C01318=2036.464500,116.962000,-461.388800,-176.322032,-0.120321,-90.000210
C01319=2037.931200,116.962000,-461.158000,-176.322032,-0.120321,-90.000210
C01320=2041.746400,116.962000,-461.186100,-176.322032,-0.120321,-90.000210
C01321=2042.791200,116.962000,-462.109500,-176.322032,-0.120321,-90.000210
C01322=2046.669400,116.962000,-461.572000,-176.322032,-0.120321,-90.000210
C01323=2047.372600,116.962000,-461.209700,-176.322032,-0.120321,-90.000210
C01324=2051.683300,116.962000,-461.572800,-176.322032,-0.120321,-90.000210
C01325=2052.215000,116.962000,-461.119800,-176.322032,-0.120321,-90.000210
C01326=2053.341500,116.962000,-460.750600,-176.322032,-0.120321,-90.000210
C01327=2055.969200,116.962000,-461.503000,-176.322032,-0.120321,-90.000210
C01328=2057.527000,116.962000,-461.105400,-176.322032,-0.120321,-90.000210
C01329=2061.172200,116.962000,-461.573500,-176.322032,-0.120321,-90.000210
C01330=2062.439400,116.962000,-461.558500,-176.322032,-0.120321,-90.000210
C01331=2065.572800,116.962000,-461.680800,-176.322032,-0.120321,-90.000210
C01332=2067.063000,116.962000,-461.000200,-176.322032,-0.120321,-90.000210
C01333=2068.716200,116.962000,-461.083200,-176.322032,-0.120321,-90.000210
C01334=2071.053200,116.962000,-461.213900,-176.322032,-0.120321,-90.000210
C01335=2072.506400,116.962000,-461.300800,-176.322032,-0.120321,-90.000210
C01336=2074.891000,116.962000,-461.196800,-176.322032,-0.120321,-90.000210
C01337=2076.394800,116.962000,-460.759700,-176.322032,-0.120321,-90.000210
C01338=2078.471600,116.962000,-461.086200,-176.322032,-0.120321,-90.000210
C01339=2081.057100,116.962000,-461.349300,-176.322032,-0.120321,-90.000210
C01340=2082.319500,116.962000,-460.447100,-176.322032,-0.120321,-90.000210
C01341=2083.837500,116.962000,-461.092800,-176.322032,-0.120321,-90.000210
C01342=2086.755400,116.962000,-460.397000,-176.322032,-0.120321,-90.000210
C01343=2087.830400,116.962000,-460.548500,-176.322032,-0.120321,-90.000210
C01344=2091.095200,116.962000,-460.597700,-176.322032,-0.120321,-90.000210
C01345=2091.982300,116.962000,-460.859600,-176.322032,-0.120321,-90.000210
C01346=2095.305000,116.962000,-460.944600,-176.322032,-0.120321,-90.000210
C01347=2096.287900,116.962000,-460.453100,-176.322032,-0.120321,-90.000210
C01348=2100.115300,116.962000,-460.344000,-176.322032,-0.120321,-90.000210
C01349=2101.997500,116.962000,-459.946600,-176.322032,-0.120321,-90.000210
C01350=2105.324200,116.962000,-459.866500,-176.322032,-0.120321,-90.000210
C01351=2107.229200,116.962000,-459.869200,-176.322032,-0.120321,-90.000210
C01352=2110.594800,116.962000,-459.783900,-176.322032,-0.120321,-90.000210
C01353=2112.130300,116.962000,-459.809200,-176.322032,-0.120321,-90.000210
C01354=2116.276900,116.962000,-459.632100,-176.322032,-0.120321,-90.000210
C01355=2116.927300,116.962000,-459.418100,-176.322032,-0.120321,-90.000210
C01356=2120.552400,116.962000,-459.569000,-176.322032,-0.120321,-90.000210
C01357=2121.891800,116.962000,-459.359100,-176.322032,-0.120321,-90.000210
C01358=2125.448600,116.962000,-458.749300,-176.322032,-0.120321,-90.000210
C01359=2126.425900,116.962000,-458.730400,-176.322032,-0.120321,-90.000210
C01360=2130.843800,116.962000,-458.929300,-176.322032,-0.120321,-90.000210
C01361=2131.792200,116.962000,-458.786400,-176.322032,-0.120321,-90.000210
C01362=2136.497100,116.962000,-458.117400,-176.322032,-0.120321,-90.000210
C01363=2137.873200,116.962000,-458.357900,-176.322032,-0.120321,-90.000210
C01364=2141.381500,116.962000,-458.142600,-176.322032,-0.120321,-90.000210
C01365=2142.294300,116.962000,-457.951200,-176.322032,-0.120321,-90.000210
C01366=2144.907900,116.962000,-457.571500,-176.322032,-0.120321,-90.000210
C01367=2146.803600,116.962000,-457.969600,-176.322032,-0.120321,-90.000210
C01368=2150.305000,116.962000,-457.602500,-176.322032,-0.120321,-90.000210
C01369=2151.528700,116.962000,-457.480600,-176.322032,-0.120321,-90.000210
C01370=2155.429600,116.962000,-457.270200,-176.322032,-0.120321,-90.000210
C01371=2157.099200,116.962000,-457.023000,-176.322032,-0.120321,-90.000210
C01372=2160.581800,116.962000,-457.022500,-176.322032,-0.120321,-90.000210
C01373=2161.665200,116.962000,-457.050900,-176.322032,-0.120321,-90.000210
C01374=2166.487200,116.962000,-456.987300,-176.322032,-0.120321,-90.000210
C01375=2167.020300,116.962000,-456.749000,-176.322032,-0.120321,-90.000210
C01376=2171.823100,116.962000,-456.380100,-176.322032,-0.120321,-90.000210
C01377=2172.384000,116.962000,-456.372000,-176.322032,-0.120321,-90.000210
C01378=2176.071000,116.962000,-456.088800,-176.322032,-0.120321,-90.000210
C01379=2176.860800,116.962000,-456.069700,-176.322032,-0.120321,-90.000210
C01380=2178.404500,116.962000,-455.836200,-176.322032,-0.120321,-90.000210
C01381=2180.545900,116.962000,-456.078600,-176.322032,-0.120321,-90.000210
C01382=2181.385200,116.962000,-455.836400,-176.322032,-0.120321,-90.000210
C01383=2182.434900,116.962000,-455.383400,-176.322032,-0.120321,-90.000210
C01384=2183.123400,116.962000,-456.497400,-176.322032,-0.120321,-90.000210
C01385=2186.978500,116.962000,-454.141500,-176.322032,-0.120321,-90.000210
C01386=2187.489500,116.962000,-454.835800,-176.322032,-0.120321,-90.000210
C01387=2190.500600,116.962000,-454.234000,-176.322032,-0.120321,-90.000210
C01388=2187.460800,66.962000,-454.621100,-176.322032,-0.120321,-90.000210
C01389=2186.546200,66.962000,-454.703500,-176.322032,-0.120321,-90.000210
C01390=2183.293200,66.962000,-454.886900,-176.322032,-0.120321,-90.000210
C01391=2182.144700,66.962000,-455.103300,-176.322032,-0.120321,-90.000210
C01392=2179.703900,66.962000,-455.685400,-176.322032,-0.120321,-90.000210
C01393=2177.868100,66.962000,-455.661700,-176.322032,-0.120321,-90.000210
C01394=2176.413500,66.962000,-456.269000,-176.322032,-0.120321,-90.000210
C01395=2174.746100,66.962000,-455.981100,-176.322032,-0.120321,-90.000210
C01396=2172.146300,66.962000,-456.415800,-176.322032,-0.120321,-90.000210
C01397=2170.888100,66.962000,-456.236600,-176.322032,-0.120321,-90.000210
C01398=2167.524500,66.962000,-456.615100,-176.322032,-0.120321,-90.000210
C01399=2166.381300,66.962000,-456.924300,-176.322032,-0.120321,-90.000210
C01400=2162.140600,66.962000,-456.879000,-176.322032,-0.120321,-90.000210
C01401=2160.998700,66.962000,-457.154200,-176.322032,-0.120321,-90.000210
C01402=2157.715600,66.962000,-457.164000,-176.322032,-0.120321,-90.000210
C01403=2156.473800,66.962000,-457.185800,-176.322032,-0.120321,-90.000210
C01404=2152.943600,66.962000,-457.775400,-176.322032,-0.120321,-90.000210
C01405=2151.910000,66.962000,-457.828300,-176.322032,-0.120321,-90.000210
C01406=2147.641800,66.962000,-458.108900,-176.322032,-0.120321,-90.000210
C01407=2145.923200,66.962000,-458.251300,-176.322032,-0.120321,-90.000210
C01408=2142.640500,66.962000,-458.570300,-176.322032,-0.120321,-90.000210
C01409=2141.323600,66.962000,-458.433500,-176.322032,-0.120321,-90.000210
C01410=2137.209300,66.962000,-458.700300,-176.322032,-0.120321,-90.000210
C01411=2136.524600,66.962000,-458.900000,-176.322032,-0.120321,-90.000210
C01412=2132.513800,66.962000,-458.772000,-176.322032,-0.120321,-90.000210
C01413=2130.736700,66.962000,-459.053600,-176.322032,-0.120321,-90.000210
C01414=2126.998500,66.962000,-458.996300,-176.322032,-0.120321,-90.000210
C01415=2125.408700,66.962000,-459.180700,-176.322032,-0.120321,-90.000210
C01416=2122.103200,66.962000,-459.050100,-176.322032,-0.120321,-90.000210
C01417=2121.398500,66.962000,-459.543000,-176.322032,-0.120321,-90.000210
C01418=2117.274100,66.962000,-459.915900,-176.322032,-0.120321,-90.000210
C01419=2116.625200,66.962000,-459.803600,-176.322032,-0.120321,-90.000210
C01420=2112.741400,66.962000,-460.134900,-176.322032,-0.120321,-90.000210
C01421=2111.498800,66.962000,-459.901200,-176.322032,-0.120321,-90.000210
C01422=2107.364300,66.962000,-460.372100,-176.322032,-0.120321,-90.000210
C01423=2106.113400,66.962000,-460.172300,-176.322032,-0.120321,-90.000210
C01424=2102.272500,66.962000,-460.391900,-176.322032,-0.120321,-90.000210
C01425=2101.374900,66.962000,-460.360100,-176.322032,-0.120321,-90.000210
C01426=2097.664400,66.962000,-460.540100,-176.322032,-0.120321,-90.000210
C01427=2096.357700,66.962000,-460.242400,-176.322032,-0.120321,-90.000210
C01428=2092.441200,66.962000,-460.698100,-176.322032,-0.120321,-90.000210
C01429=2091.853500,66.962000,-460.725400,-176.322032,-0.120321,-90.000210
C01430=2090.580900,66.962000,-460.670300,-176.322032,-0.120321,-90.000210
C01431=2087.672500,66.962000,-460.988000,-176.322032,-0.120321,-90.000210
C01432=2086.891600,66.962000,-461.118100,-176.322032,-0.120321,-90.000210
C01433=2085.763200,66.962000,-461.022000,-176.322032,-0.120321,-90.000210
C01434=2082.853700,66.962000,-461.325900,-176.322032,-0.120321,-90.000210
C01435=2081.388800,66.962000,-461.142700,-176.322032,-0.120321,-90.000210
C01436=2078.659000,66.962000,-460.798200,-176.322032,-0.120321,-90.000210
C01437=2077.339900,66.962000,-460.592800,-176.322032,-0.120321,-90.000210
C01438=2076.693000,66.962000,-460.982800,-176.322032,-0.120321,-90.000210
C01439=2075.624700,66.962000,-460.685400,-176.322032,-0.120321,-90.000210
C01440=2072.957600,66.962000,-461.172700,-176.322032,-0.120321,-90.000210
C01441=2071.852900,66.962000,-461.354700,-176.322032,-0.120321,-90.000210
C01442=2068.101300,66.962000,-460.816200,-176.322032,-0.120321,-90.000210
C01443=2067.089500,66.962000,-461.221500,-176.322032,-0.120321,-90.000210
C01444=2066.067700,66.962000,-461.312200,-176.322032,-0.120321,-90.000210
C01445=2061.935200,66.962000,-461.790200,-176.322032,-0.120321,-90.000210
C01446=2061.303500,66.962000,-461.490200,-176.322032,-0.120321,-90.000210
C01447=2057.096300,66.962000,-461.766500,-176.322032,-0.120321,-90.000210
C01448=2056.220800,66.962000,-461.730600,-176.322032,-0.120321,-90.000210
C01449=2052.714800,66.962000,-461.821300,-176.322032,-0.120321,-90.000210
C01450=2051.615100,66.962000,-461.465000,-176.322032,-0.120321,-90.000210
C01451=2047.197100,66.962000,-462.015900,-176.322032,-0.120321,-90.000210
C01452=2046.669800,66.962000,-461.560700,-176.322032,-0.120321,-90.000210
C01453=2042.419200,66.962000,-461.438300,-176.322032,-0.120321,-90.000210
C01454=2041.321400,66.962000,-461.722900,-176.322032,-0.120321,-90.000210
C01455=2037.944000,66.962000,-461.891700,-176.322032,-0.120321,-90.000210
C01456=2036.779200,66.962000,-461.544600,-176.322032,-0.120321,-90.000210
C01457=2032.602700,66.962000,-461.671200,-176.322032,-0.120321,-90.000210
C01458=2032.128600,66.962000,-462.191800,-176.322032,-0.120321,-90.000210
C01459=2027.146500,66.962000,-461.876500,-176.322032,-0.120321,-90.000210
C01460=2026.533400,66.962000,-462.228000,-176.322032,-0.120321,-90.000210
C01461=2022.435100,66.962000,-462.037800,-176.322032,-0.120321,-90.000210
C01462=2021.425300,66.962000,-461.958100,-176.322032,-0.120321,-90.000210
C01463=2017.590500,66.962000,-461.902400,-176.322032,-0.120321,-90.000210
C01464=2017.006800,66.962000,-461.655800,-176.322032,-0.120321,-90.000210
C01465=2012.532100,66.962000,-462.194700,-176.322032,-0.120321,-90.000210
C01466=2012.154700,66.962000,-462.076800,-176.322032,-0.120321,-90.000210
C01467=2007.660100,66.962000,-462.120400,-176.322032,-0.120321,-90.000210
C01468=2006.639900,66.962000,-461.912600,-176.322032,-0.120321,-90.000210
C01469=2002.362600,66.962000,-462.269100,-176.322032,-0.120321,-90.000210
C01470=2001.731700,66.962000,-461.761800,-176.322032,-0.120321,-90.000210
C01471=1997.924200,66.962000,-462.524400,-176.322032,-0.120321,-90.000210
C01472=1996.573400,66.962000,-462.089000,-176.322032,-0.120321,-90.000210
C01473=1991.968800,66.962000,-462.726500,-176.322032,-0.120321,-90.000210
C01474=1991.298200,66.962000,-461.843300,-176.322032,-0.120321,-90.000210
C01475=1987.289200,66.962000,-461.999200,-176.322032,-0.120321,-90.000210
C01476=1986.814500,66.962000,-462.667300,-176.322032,-0.120321,-90.000210
C01477=1982.523900,66.962000,-462.299700,-176.322032,-0.120321,-90.000210
C01478=1981.365600,66.962000,-462.426300,-176.322032,-0.120321,-90.000210
C01479=1977.592200,66.962000,-462.407800,-176.322032,-0.120321,-90.000210
C01480=1976.591300,66.962000,-462.624200,-176.322032,-0.120321,-90.000210
C01481=1972.053400,66.962000,-462.402800,-176.322032,-0.120321,-90.000210
C01482=1971.187300,66.962000,-462.283800,-176.322032,-0.120321,-90.000210
C01483=1967.390600,66.962000,-462.352500,-176.322032,-0.120321,-90.000210
C01484=1966.281000,66.962000,-462.481700,-176.322032,-0.120321,-90.000210
C01485=1962.364900,66.962000,-462.681000,-176.322032,-0.120321,-90.000210
C01486=1961.526700,66.962000,-462.462900,-176.322032,-0.120321,-90.000210
C01487=1957.191000,66.962000,-462.718900,-176.322032,-0.120321,-90.000210
C01488=1956.508800,66.962000,-463.070800,-176.322032,-0.120321,-90.000210
C01489=1952.212400,66.962000,-462.659600,-176.322032,-0.120321,-90.000210
C01490=1951.195700,66.962000,-462.740300,-176.322032,-0.120321,-90.000210
C01491=1947.001000,66.962000,-462.695400,-176.322032,-0.120321,-90.000210
C01492=1946.188100,66.962000,-462.863100,-176.322032,-0.120321,-90.000210
C01493=1942.202500,66.962000,-462.673200,-176.322032,-0.120321,-90.000210
C01494=1941.556900,66.962000,-462.520400,-176.322032,-0.120321,-90.000210
C01495=1936.692100,66.962000,-462.898600,-176.322032,-0.120321,-90.000210
C01496=1936.108700,66.962000,-462.734800,-176.322032,-0.120321,-90.000210
C01497=1931.690400,66.962000,-462.982900,-176.322032,-0.120321,-90.000210
C01498=1930.845700,66.962000,-462.918100,-176.322032,-0.120321,-90.000210
C01499=1927.277900,66.962000,-463.021300,-176.322032,-0.120321,-90.000210
C01500=1926.380500,66.962000,-462.614200,-176.322032,-0.120321,-90.000210
C01501=1922.306400,66.962000,-462.887700,-176.322032,-0.120321,-90.000210
C01502=1920.906400,66.962000,-462.932600,-176.322032,-0.120321,-90.000210
C01503=1917.431300,66.962000,-462.524900,-176.322032,-0.120321,-90.000210
C01504=1916.235300,66.962000,-462.501100,-176.322032,-0.120321,-90.000210
C01505=1912.599900,66.962000,-462.603100,-176.322032,-0.120321,-90.000210
C01506=1910.569000,66.962000,-462.776000,-176.322032,-0.120321,-90.000210
C01507=1906.891700,66.962000,-462.472500,-176.322032,-0.120321,-90.000210
C01508=1905.947500,66.962000,-462.866000,-176.322032,-0.120321,-90.000210
C01509=1901.562100,66.962000,-462.900500,-176.322032,-0.120321,-90.000210
C01510=1901.024600,66.962000,-462.765600,-176.322032,-0.120321,-90.000210
C01511=1896.366700,66.962000,-462.571200,-176.322032,-0.120321,-90.000210
C01512=1895.945300,66.962000,-462.685500,-176.322032,-0.120321,-90.000210
C01513=1892.072500,66.962000,-462.600000,-176.322032,-0.120321,-90.000210
C01514=1887.540100,66.962000,-462.340500,-176.322032,-0.120321,-90.000210
C01515=1887.060500,66.962000,-462.329200,-176.322032,-0.120321,-90.000210
C01516=1883.578900,66.962000,-461.818100,-176.322032,-0.120321,-90.000210
C01517=1881.534600,66.962000,-462.313800,-176.322032,-0.120321,-90.000210
C01518=1877.920400,66.962000,-462.348400,-176.322032,-0.120321,-90.000210
C01519=1877.012100,66.962000,-462.257500,-176.322032,-0.120321,-90.000210
C01520=1873.176100,66.962000,-462.090200,-176.322032,-0.120321,-90.000210
C01521=1871.982100,66.962000,-461.820500,-176.322032,-0.120321,-90.000210
C01522=1867.738500,66.962000,-461.710300,-176.322032,-0.120321,-90.000210
C01523=1866.173600,66.962000,-461.878900,-176.322032,-0.120321,-90.000210
C01524=1862.125600,66.962000,-461.492800,-176.322032,-0.120321,-90.000210
C01525=1861.102200,66.962000,-461.128300,-176.322032,-0.120321,-90.000210
C01526=1858.018300,66.962000,-461.616900,-176.322032,-0.120321,-90.000210
C01527=1856.295800,66.962000,-460.869200,-176.322032,-0.120321,-90.000210
C01528=1854.579600,66.962000,-461.148100,-176.322032,-0.120321,-90.000210
C01529=1852.507200,66.962000,-461.287100,-176.322032,-0.120321,-90.000210
C01530=1851.208800,66.962000,-461.126800,-176.322032,-0.120321,-90.000210
C01531=1849.888800,66.962000,-460.848500,-176.322032,-0.120321,-90.000210
C01532=1847.630900,66.962000,-460.811400,-176.322032,-0.120321,-90.000210
C01533=1846.477100,66.962000,-460.758100,-176.322032,-0.120321,-90.000210
C01534=1844.129100,66.962000,-460.736500,-176.322032,-0.120321,-90.000210
C01535=1841.569400,66.962000,-460.494100,-176.322032,-0.120321,-90.000210
C01536=1837.832100,66.962000,-460.286000,-176.322032,-0.120321,-90.000210
C01537=1836.209500,66.962000,-460.222500,-176.322032,-0.120321,-90.000210
C01538=1832.383000,66.962000,-460.143800,-176.322032,-0.120321,-90.000210
C01539=1831.289100,66.962000,-459.907100,-176.322032,-0.120321,-90.000210
C01540=1827.422300,66.962000,-459.786000,-176.322032,-0.120321,-90.000210
C01541=1826.770000,66.962000,-459.789300,-176.322032,-0.120321,-90.000210
C01542=1822.655900,66.962000,-459.121000,-176.322032,-0.120321,-90.000210
C01543=1822.031800,66.962000,-459.340400,-176.322032,-0.120321,-90.000210
C01544=1817.166700,66.962000,-458.933700,-176.322032,-0.120321,-90.000210
C01545=1815.927200,66.962000,-458.829300,-176.322032,-0.120321,-90.000210
C01546=1812.134000,66.962000,-458.724000,-176.322032,-0.120321,-90.000210
C01547=1811.547400,66.962000,-458.669000,-176.322032,-0.120321,-90.000210
C01548=1807.539800,66.962000,-458.085800,-176.322032,-0.120321,-90.000210
C01549=1806.155800,66.962000,-458.104200,-176.322032,-0.120321,-90.000210
C01550=1802.582800,66.962000,-457.791500,-176.322032,-0.120321,-90.000210
C01551=1802.038800,66.962000,-457.763400,-176.322032,-0.120321,-90.000210
C01552=1797.104900,66.962000,-456.696100,-176.322032,-0.120321,-90.000210
C01553=1800.853000,16.962000,-457.600400,-176.322032,-0.120321,-90.000210
C01554=1801.833400,16.962000,-457.702300,-176.322032,-0.120321,-90.000210
C01555=1805.690500,16.962000,-457.850100,-176.322032,-0.120321,-90.000210
C01556=1806.955100,16.962000,-458.128800,-176.322032,-0.120321,-90.000210
C01557=1810.171000,16.962000,-458.514800,-176.322032,-0.120321,-90.000210
C01558=1812.204800,16.962000,-458.248700,-176.322032,-0.120321,-90.000210
C01559=1815.347500,16.962000,-458.808000,-176.322032,-0.120321,-90.000210
C01560=1816.625200,16.962000,-458.841700,-176.322032,-0.120321,-90.000210
C01561=1819.689800,16.962000,-458.842800,-176.322032,-0.120321,-90.000210
C01562=1821.724100,16.962000,-459.142000,-176.322032,-0.120321,-90.000210
C01563=1825.694700,16.962000,-459.364300,-176.322032,-0.120321,-90.000210
C01564=1826.988700,16.962000,-459.139000,-176.322032,-0.120321,-90.000210
C01565=1830.989300,16.962000,-460.055400,-176.322032,-0.120321,-90.000210
C01566=1832.117900,16.962000,-459.845800,-176.322032,-0.120321,-90.000210
C01567=1835.624600,16.962000,-460.233700,-176.322032,-0.120321,-90.000210
C01568=1836.819800,16.962000,-460.243900,-176.322032,-0.120321,-90.000210
C01569=1840.600200,16.962000,-460.486000,-176.322032,-0.120321,-90.000210
C01570=1841.684100,16.962000,-460.100000,-176.322032,-0.120321,-90.000210
C01571=1842.855500,16.962000,-460.996600,-176.322032,-0.120321,-90.000210
C01572=1846.207800,16.962000,-460.276800,-176.322032,-0.120321,-90.000210
C01573=1847.787400,16.962000,-460.089300,-176.322032,-0.120321,-90.000210
C01574=1850.604200,16.962000,-460.507100,-176.322032,-0.120321,-90.000210
C01575=1851.898200,16.962000,-460.731700,-176.322032,-0.120321,-90.000210
C01576=1853.812100,16.962000,-460.957800,-176.322032,-0.120321,-90.000210
C01577=1856.051100,16.962000,-461.225800,-176.322032,-0.120321,-90.000210
C01578=1856.992500,16.962000,-460.979300,-176.322032,-0.120321,-90.000210
C01579=1860.909800,16.962000,-460.744600,-176.322032,-0.120321,-90.000210
C01580=1862.312000,16.962000,-461.462200,-176.322032,-0.120321,-90.000210
C01581=1863.680400,16.962000,-461.168200,-176.322032,-0.120321,-90.000210
C01582=1867.087300,16.962000,-461.817800,-176.322032,-0.120321,-90.000210
C01583=1868.078400,16.962000,-460.823400,-176.322032,-0.120321,-90.000210
C01584=1871.197200,16.962000,-462.036800,-176.322032,-0.120321,-90.000210
C01585=1871.740000,16.962000,-461.205200,-176.322032,-0.120321,-90.000210
C01586=1876.026500,16.962000,-461.728400,-176.322032,-0.120321,-90.000210
C01587=1876.941400,16.962000,-461.824400,-176.322032,-0.120321,-90.000210
C01588=1879.389400,16.962000,-461.693700,-176.322032,-0.120321,-90.000210
C01589=1882.239000,16.962000,-461.511900,-176.322032,-0.120321,-90.000210
C01590=1883.592600,16.962000,-461.739600,-176.322032,-0.120321,-90.000210
C01591=1886.781000,16.962000,-462.128300,-176.322032,-0.120321,-90.000210
C01592=1888.118700,16.962000,-461.470900,-176.322032,-0.120321,-90.000210
C01593=1892.080400,16.962000,-462.546100,-176.322032,-0.120321,-90.000210
C01594=1893.191100,16.962000,-462.370500,-176.322032,-0.120321,-90.000210
C01595=1897.094800,16.962000,-462.092100,-176.322032,-0.120321,-90.000210
C01596=1898.386500,16.962000,-462.636900,-176.322032,-0.120321,-90.000210
C01597=1901.138700,16.962000,-462.159200,-176.322032,-0.120321,-90.000210
C01598=1902.847400,16.962000,-461.680000,-176.322032,-0.120321,-90.000210
C01599=1906.862100,16.962000,-462.063600,-176.322032,-0.120321,-90.000210
C01600=1907.774900,16.962000,-461.771400,-176.322032,-0.120321,-90.000210
C01601=1911.590400,16.962000,-461.818300,-176.322032,-0.120321,-90.000210
C01602=1916.132700,16.962000,-461.555400,-176.322032,-0.120321,-90.000210
C01603=1917.627600,16.962000,-462.395700,-176.322032,-0.120321,-90.000210
C01604=1920.150200,16.962000,-461.852400,-176.322032,-0.120321,-90.000210
C01605=1922.503800,16.962000,-462.108200,-176.322032,-0.120321,-90.000210
C01606=1925.787300,16.962000,-462.559600,-176.322032,-0.120321,-90.000210
C01607=1927.580300,16.962000,-462.489900,-176.322032,-0.120321,-90.000210
C01608=1930.883000,16.962000,-462.130700,-176.322032,-0.120321,-90.000210
C01609=1932.180200,16.962000,-462.049300,-176.322032,-0.120321,-90.000210
C01610=1936.098200,16.962000,-461.733900,-176.322032,-0.120321,-90.000210
C01611=1937.465400,16.962000,-461.859600,-176.322032,-0.120321,-90.000210
C01612=1940.869700,16.962000,-461.667300,-176.322032,-0.120321,-90.000210
C01613=1941.947000,16.962000,-461.985100,-176.322032,-0.120321,-90.000210
C01614=1946.026000,16.962000,-461.537600,-176.322032,-0.120321,-90.000210
C01615=1947.031900,16.962000,-460.749300,-176.322032,-0.120321,-90.000210
C01616=1950.520700,16.962000,-462.488400,-176.322032,-0.120321,-90.000210
C01617=1951.508200,16.962000,-462.017400,-176.322032,-0.120321,-90.000210
C01618=1953.630300,16.962000,-460.907700,-176.322032,-0.120321,-90.000210
C01619=1956.666900,16.962000,-461.810100,-176.322032,-0.120321,-90.000210
C01620=1958.240000,16.962000,-461.138900,-176.322032,-0.120321,-90.000210
C01621=1961.763500,16.962000,-461.648500,-176.322032,-0.120321,-90.000210
C01622=1962.592900,16.962000,-461.669800,-176.322032,-0.120321,-90.000210
C01623=1966.715800,16.962000,-462.226500,-176.322032,-0.120321,-90.000210
C01624=1967.742300,16.962000,-461.460300,-176.322032,-0.120321,-90.000210
C01625=1971.291200,16.962000,-461.488500,-176.322032,-0.120321,-90.000210
C01626=1972.357700,16.962000,-461.185800,-176.322032,-0.120321,-90.000210
C01627=1976.644300,16.962000,-461.744300,-176.322032,-0.120321,-90.000210
C01628=1977.172500,16.962000,-461.461900,-176.322032,-0.120321,-90.000210
C01629=1981.055200,16.962000,-462.223500,-176.322032,-0.120321,-90.000210
C01630=1982.924200,16.962000,-461.277500,-176.322032,-0.120321,-90.000210
C01631=1985.903600,16.962000,-461.979500,-176.322032,-0.120321,-90.000210
C01632=1987.027800,16.962000,-462.156500,-176.322032,-0.120321,-90.000210
C01633=1990.724500,16.962000,-461.454900,-176.322032,-0.120321,-90.000210
C01634=1991.847500,16.962000,-461.089000,-176.322032,-0.120321,-90.000210
C01635=1992.300200,16.962000,-461.929400,-176.322032,-0.120321,-90.000210
C01636=1995.887600,16.962000,-461.863300,-176.322032,-0.120321,-90.000210
C01637=1997.305400,16.962000,-462.410800,-176.322032,-0.120321,-90.000210
C01638=2001.335200,16.962000,-461.762900,-176.322032,-0.120321,-90.000210
C01639=2001.915900,16.962000,-461.490300,-176.322032,-0.120321,-90.000210
C01640=2003.087800,16.962000,-460.638700,-176.322032,-0.120321,-90.000210
C01641=2005.703100,16.962000,-462.013900,-176.322032,-0.120321,-90.000210
C01642=2007.016400,16.962000,-461.067600,-176.322032,-0.120321,-90.000210
C01643=2010.670700,16.962000,-461.084200,-176.322032,-0.120321,-90.000210
C01644=2011.764900,16.962000,-461.877300,-176.322032,-0.120321,-90.000210
C01645=2014.884300,16.962000,-460.917300,-176.322032,-0.120321,-90.000210
C01646=2017.022900,16.962000,-461.622600,-176.322032,-0.120321,-90.000210
C01647=2018.108600,16.962000,-461.481100,-176.322032,-0.120321,-90.000210
C01648=2020.072500,16.962000,-461.472200,-176.322032,-0.120321,-90.000210
C01649=2021.496700,16.962000,-461.126300,-176.322032,-0.120321,-90.000210
C01650=2022.573700,16.962000,-461.597500,-176.322032,-0.120321,-90.000210
C01651=2025.356300,16.962000,-460.919900,-176.322032,-0.120321,-90.000210
C01652=2027.389200,16.962000,-460.852400,-176.322032,-0.120321,-90.000210
C01653=2028.101900,16.962000,-461.298000,-176.322032,-0.120321,-90.000210
C01654=2031.703300,16.962000,-460.626700,-176.322032,-0.120321,-90.000210
C01655=2032.902100,16.962000,-461.367200,-176.322032,-0.120321,-90.000210
C01656=2035.802300,16.962000,-460.830300,-176.322032,-0.120321,-90.000210
C01657=2037.079400,16.962000,-460.852900,-176.322032,-0.120321,-90.000210
C01658=2038.174900,16.962000,-460.664800,-176.322032,-0.120321,-90.000210
C01659=2041.615300,16.962000,-461.220900,-176.322032,-0.120321,-90.000210
C01660=2042.295400,16.962000,-461.025900,-176.322032,-0.120321,-90.000210
C01661=2046.640700,16.962000,-460.294900,-176.322032,-0.120321,-90.000210
C01662=2047.090900,16.962000,-461.310000,-176.322032,-0.120321,-90.000210
C01663=2048.126700,16.962000,-461.431700,-176.322032,-0.120321,-90.000210
C01664=2051.137100,16.962000,-461.425400,-176.322032,-0.120321,-90.000210
C01665=2052.144900,16.962000,-460.788200,-176.322032,-0.120321,-90.000210
C01666=2053.757600,16.962000,-460.715100,-176.322032,-0.120321,-90.000210
C01667=2055.647100,16.962000,-461.029500,-176.322032,-0.120321,-90.000210
C01668=2056.837400,16.962000,-460.592600,-176.322032,-0.120321,-90.000210
C01669=2058.334000,16.962000,-460.769100,-176.322032,-0.120321,-90.000210
C01670=2060.286200,16.962000,-460.650500,-176.322032,-0.120321,-90.000210
C01671=2061.744300,16.962000,-461.198600,-176.322032,-0.120321,-90.000210
C01672=2063.209100,16.962000,-460.755400,-176.322032,-0.120321,-90.000210
C01673=2065.833000,16.962000,-461.205700,-176.322032,-0.120321,-90.000210
C01674=2067.142800,16.962000,-461.197800,-176.322032,-0.120321,-90.000210
C01675=2068.505600,16.962000,-461.026200,-176.322032,-0.120321,-90.000210
C01676=2071.236500,16.962000,-460.349100,-176.322032,-0.120321,-90.000210
C01677=2072.661000,16.962000,-460.841900,-176.322032,-0.120321,-90.000210
C01678=2073.832100,16.962000,-460.585700,-176.322032,-0.120321,-90.000210
C01679=2076.319000,16.962000,-460.985400,-176.322032,-0.120321,-90.000210
C01680=2077.381000,16.962000,-460.675300,-176.322032,-0.120321,-90.000210
C01681=2080.891400,16.962000,-460.532900,-176.322032,-0.120321,-90.000210
C01682=2081.908100,16.962000,-460.506000,-176.322032,-0.120321,-90.000210
C01683=2086.379400,16.962000,-460.673900,-176.322032,-0.120321,-90.000210
C01684=2087.105400,16.962000,-460.580200,-176.322032,-0.120321,-90.000210
C01685=2089.705100,16.962000,-460.365500,-176.322032,-0.120321,-90.000210
C01686=2091.207800,16.962000,-459.880700,-176.322032,-0.120321,-90.000210
C01687=2092.153100,16.962000,-461.155000,-176.322032,-0.120321,-90.000210
C01688=2096.423800,16.962000,-459.934900,-176.322032,-0.120321,-90.000210
C01689=2098.040400,16.962000,-460.150100,-176.322032,-0.120321,-90.000210
C01690=2101.854200,16.962000,-460.057700,-176.322032,-0.120321,-90.000210
C01691=2103.156700,16.962000,-459.863300,-176.322032,-0.120321,-90.000210
C01692=2107.026800,16.962000,-460.274800,-176.322032,-0.120321,-90.000210
C01693=2108.397300,16.962000,-459.836500,-176.322032,-0.120321,-90.000210
C01694=2111.487600,16.962000,-459.859600,-176.322032,-0.120321,-90.000210
C01695=2112.805300,16.962000,-459.587300,-176.322032,-0.120321,-90.000210
C01696=2116.598800,16.962000,-459.175700,-176.322032,-0.120321,-90.000210
C01697=2117.416700,16.962000,-459.383000,-176.322032,-0.120321,-90.000210
C01698=2121.547300,16.962000,-458.800000,-176.322032,-0.120321,-90.000210
C01699=2123.457300,16.962000,-458.872100,-176.322032,-0.120321,-90.000210
C01700=2126.573300,16.962000,-458.699900,-176.322032,-0.120321,-90.000210
C01701=2128.269900,16.962000,-458.632900,-176.322032,-0.120321,-90.000210
C01702=2132.065400,16.962000,-458.759400,-176.322032,-0.120321,-90.000210
C01703=2135.214800,16.962000,-458.605800,-176.322032,-0.120321,-90.000210
C01704=2137.412900,16.962000,-458.714700,-176.322032,-0.120321,-90.000210
C01705=2140.859300,16.962000,-458.398500,-176.322032,-0.120321,-90.000210
C01706=2142.455100,16.962000,-458.453300,-176.322032,-0.120321,-90.000210
C01707=2145.178200,16.962000,-458.252400,-176.322032,-0.120321,-90.000210
C01708=2146.847400,16.962000,-457.833500,-176.322032,-0.120321,-90.000210
C01709=2150.225600,16.962000,-458.008400,-176.322032,-0.120321,-90.000210
C01710=2151.796600,16.962000,-457.562300,-176.322032,-0.120321,-90.000210
C01711=2156.035700,16.962000,-457.211800,-176.322032,-0.120321,-90.000210
C01712=2157.040800,16.962000,-457.575900,-176.322032,-0.120321,-90.000210
C01713=2160.864800,16.962000,-456.858600,-176.322032,-0.120321,-90.000210
C01714=2162.183900,16.962000,-457.012700,-176.322032,-0.120321,-90.000210
C01715=2165.849300,16.962000,-456.622500,-176.322032,-0.120321,-90.000210
C01716=2166.839300,16.962000,-456.782400,-176.322032,-0.120321,-90.000210
C01717=2171.345200,16.962000,-456.357400,-176.322032,-0.120321,-90.000210
C01718=2172.133800,16.962000,-456.245200,-176.322032,-0.120321,-90.000210
C01719=2173.733600,16.962000,-455.771000,-176.322032,-0.120321,-90.000210
C01720=2176.308000,16.962000,-456.085000,-176.322032,-0.120321,-90.000210
C01721=2177.318900,16.962000,-456.012400,-176.322032,-0.120321,-90.000210
C01722=2178.967000,16.962000,-456.161600,-176.322032,-0.120321,-90.000210
C01723=2182.520600,16.962000,-455.315500,-176.322032,-0.120321,-90.000210
C01724=2183.036800,16.962000,-455.109100,-176.322032,-0.120321,-90.000210
C01725=2186.484700,16.962000,-454.724100,-176.322032,-0.120321,-90.000210
C01726=2187.838700,-33.038000,-454.194000,-176.322032,-0.120321,-90.000210
C01727=2186.454500,-33.038000,-454.700600,-176.322032,-0.120321,-90.000210
C01728=2183.213500,-33.038000,-455.001300,-176.322032,-0.120321,-90.000210
C01729=2181.860300,-33.038000,-455.251100,-176.322032,-0.120321,-90.000210
C01730=2179.250400,-33.038000,-455.735500,-176.322032,-0.120321,-90.000210
C01731=2176.946500,-33.038000,-456.101100,-176.322032,-0.120321,-90.000210
C01732=2175.426200,-33.038000,-456.242900,-176.322032,-0.120321,-90.000210
C01733=2172.831900,-33.038000,-455.920500,-176.322032,-0.120321,-90.000210
C01734=2171.322200,-33.038000,-456.459500,-176.322032,-0.120321,-90.000210
C01735=2168.024400,-33.038000,-456.212800,-176.322032,-0.120321,-90.000210
C01736=2167.233900,-33.038000,-456.321600,-176.322032,-0.120321,-90.000210
C01737=2165.443700,-33.038000,-456.078900,-176.322032,-0.120321,-90.000210
C01738=2162.061200,-33.038000,-456.737100,-176.322032,-0.120321,-90.000210
C01739=2160.812000,-33.038000,-456.592500,-176.322032,-0.120321,-90.000210
C01740=2157.031700,-33.038000,-457.063500,-176.322032,-0.120321,-90.000210
C01741=2155.682900,-33.038000,-456.848600,-176.322032,-0.120321,-90.000210
C01742=2152.307700,-33.038000,-457.399000,-176.322032,-0.120321,-90.000210
C01743=2151.095400,-33.038000,-456.909100,-176.322032,-0.120321,-90.000210
C01744=2147.119000,-33.038000,-457.698900,-176.322032,-0.120321,-90.000210
C01745=2146.285500,-33.038000,-457.464800,-176.322032,-0.120321,-90.000210
C01746=2142.094500,-33.038000,-457.317000,-176.322032,-0.120321,-90.000210
C01747=2140.940300,-33.038000,-458.102200,-176.322032,-0.120321,-90.000210
C01748=2137.249800,-33.038000,-457.849200,-176.322032,-0.120321,-90.000210
C01749=2135.800200,-33.038000,-458.404700,-176.322032,-0.120321,-90.000210
C01750=2132.447400,-33.038000,-457.888900,-176.322032,-0.120321,-90.000210
C01751=2130.881900,-33.038000,-458.017200,-176.322032,-0.120321,-90.000210
C01752=2127.696600,-33.038000,-458.392200,-176.322032,-0.120321,-90.000210
C01753=2125.934400,-33.038000,-457.589900,-176.322032,-0.120321,-90.000210
C01754=2122.034300,-33.038000,-458.169100,-176.322032,-0.120321,-90.000210
C01755=2120.860300,-33.038000,-458.711400,-176.322032,-0.120321,-90.000210
C01756=2116.693700,-33.038000,-459.001300,-176.322032,-0.120321,-90.000210
C01757=2115.536600,-33.038000,-458.957700,-176.322032,-0.120321,-90.000210
C01758=2112.057100,-33.038000,-458.432200,-176.322032,-0.120321,-90.000210
C01759=2111.520200,-33.038000,-458.485900,-176.322032,-0.120321,-90.000210
C01760=2107.335500,-33.038000,-459.507600,-176.322032,-0.120321,-90.000210
C01761=2106.856800,-33.038000,-458.373000,-176.322032,-0.120321,-90.000210
C01762=2102.696100,-33.038000,-458.762800,-176.322032,-0.120321,-90.000210
C01763=2101.749000,-33.038000,-459.833100,-176.322032,-0.120321,-90.000210
C01764=2097.182800,-33.038000,-459.129800,-176.322032,-0.120321,-90.000210
C01765=2095.888800,-33.038000,-459.330300,-176.322032,-0.120321,-90.000210
C01766=2091.851900,-33.038000,-459.415900,-176.322032,-0.120321,-90.000210
C01767=2091.217600,-33.038000,-459.772400,-176.322032,-0.120321,-90.000210
C01768=2087.288800,-33.038000,-459.756000,-176.322032,-0.120321,-90.000210
C01769=2085.837800,-33.038000,-458.509600,-176.322032,-0.120321,-90.000210
C01770=2081.795300,-33.038000,-459.414600,-176.322032,-0.120321,-90.000210
C01771=2080.997400,-33.038000,-459.367000,-176.322032,-0.120321,-90.000210
C01772=2076.630700,-33.038000,-458.860300,-176.322032,-0.120321,-90.000210
C01773=2076.051100,-33.038000,-459.656600,-176.322032,-0.120321,-90.000210
C01774=2072.015300,-33.038000,-458.713600,-176.322032,-0.120321,-90.000210
C01775=2071.035200,-33.038000,-459.399500,-176.322032,-0.120321,-90.000210
C01776=2067.236600,-33.038000,-459.249200,-176.322032,-0.120321,-90.000210
C01777=2065.839300,-33.038000,-458.730200,-176.322032,-0.120321,-90.000210
C01778=2062.160200,-33.038000,-458.971100,-176.322032,-0.120321,-90.000210
C01779=2061.058300,-33.038000,-459.739300,-176.322032,-0.120321,-90.000210
C01780=2057.081800,-33.038000,-459.848100,-176.322032,-0.120321,-90.000210
C01781=2055.954700,-33.038000,-459.049100,-176.322032,-0.120321,-90.000210
C01782=2051.778400,-33.038000,-459.442300,-176.322032,-0.120321,-90.000210
C01783=2051.093500,-33.038000,-460.698900,-176.322032,-0.120321,-90.000210
C01784=2047.182700,-33.038000,-460.243600,-176.322032,-0.120321,-90.000210
C01785=2046.729900,-33.038000,-459.904100,-176.322032,-0.120321,-90.000210
C01786=2042.216200,-33.038000,-460.457100,-176.322032,-0.120321,-90.000210
C01787=2041.294800,-33.038000,-458.744200,-176.322032,-0.120321,-90.000210
C01788=2037.518900,-33.038000,-459.148400,-176.322032,-0.120321,-90.000210
C01789=2035.474300,-33.038000,-460.335600,-176.322032,-0.120321,-90.000210
C01790=2031.929200,-33.038000,-460.110300,-176.322032,-0.120321,-90.000210
C01791=2029.976300,-33.038000,-459.700900,-176.322032,-0.120321,-90.000210
C01792=2027.239700,-33.038000,-459.399800,-176.322032,-0.120321,-90.000210
C01793=2025.810000,-33.038000,-459.211800,-176.322032,-0.120321,-90.000210
C01794=2021.686800,-33.038000,-459.299000,-176.322032,-0.120321,-90.000210
C01795=2021.017400,-33.038000,-460.534600,-176.322032,-0.120321,-90.000210
C01796=2016.905600,-33.038000,-459.977300,-176.322032,-0.120321,-90.000210
C01797=2012.348800,-33.038000,-459.566100,-176.322032,-0.120321,-90.000210
C01798=2011.690400,-33.038000,-460.454600,-176.322032,-0.120321,-90.000210
C01799=2008.176400,-33.038000,-460.018800,-176.322032,-0.120321,-90.000210
C01800=2006.344600,-33.038000,-459.093500,-176.322032,-0.120321,-90.000210
C01801=2003.207100,-33.038000,-460.862300,-176.322032,-0.120321,-90.000210
C01802=2002.338200,-33.038000,-459.942100,-176.322032,-0.120321,-90.000210
C01803=1999.720100,-33.038000,-461.131000,-176.322032,-0.120321,-90.000210
C01804=1997.072500,-33.038000,-460.970300,-176.322032,-0.120321,-90.000210
C01805=1996.611600,-33.038000,-458.972600,-176.322032,-0.120321,-90.000210
C01806=1991.746400,-33.038000,-460.075000,-176.322032,-0.120321,-90.000210
C01807=1990.974800,-33.038000,-458.928700,-176.322032,-0.120321,-90.000210
C01808=1988.250500,-33.038000,-460.146800,-176.322032,-0.120321,-90.000210
C01809=1986.586300,-33.038000,-459.666500,-176.322032,-0.120321,-90.000210
C01810=1982.669800,-33.038000,-460.393600,-176.322032,-0.120321,-90.000210
C01811=1982.006000,-33.038000,-460.568200,-176.322032,-0.120321,-90.000210
C01812=1978.599200,-33.038000,-461.372600,-176.322032,-0.120321,-90.000210
C01813=1977.058700,-33.038000,-459.119900,-176.322032,-0.120321,-90.000210
C01814=1975.657300,-33.038000,-460.292600,-176.322032,-0.120321,-90.000210
C01815=1971.969300,-33.038000,-459.202100,-176.322032,-0.120321,-90.000210
C01816=1970.572200,-33.038000,-461.094400,-176.322032,-0.120321,-90.000210
C01817=1967.981000,-33.038000,-460.591300,-176.322032,-0.120321,-90.000210
C01818=1966.614200,-33.038000,-459.028200,-176.322032,-0.120321,-90.000210
C01819=1962.506300,-33.038000,-459.253800,-176.322032,-0.120321,-90.000210
C01820=1961.381100,-33.038000,-459.030500,-176.322032,-0.120321,-90.000210
C01821=1959.432500,-33.038000,-461.204400,-176.322032,-0.120321,-90.000210
C01822=1957.002400,-33.038000,-460.734200,-176.322032,-0.120321,-90.000210
C01823=1956.020800,-33.038000,-460.682600,-176.322032,-0.120321,-90.000210
C01824=1952.100400,-33.038000,-459.585000,-176.322032,-0.120321,-90.000210
C01825=1951.434800,-33.038000,-460.976500,-176.322032,-0.120321,-90.000210
C01826=1947.466500,-33.038000,-460.666500,-176.322032,-0.120321,-90.000210
C01827=1946.943100,-33.038000,-460.699400,-176.322032,-0.120321,-90.000210
C01828=1945.653800,-33.038000,-461.235700,-176.322032,-0.120321,-90.000210
C01829=1943.038200,-33.038000,-460.079600,-176.322032,-0.120321,-90.000210
C01830=1941.410600,-33.038000,-459.356300,-176.322032,-0.120321,-90.000210
C01831=1937.364700,-33.038000,-460.486400,-176.322032,-0.120321,-90.000210
C01832=1936.135000,-33.038000,-459.630900,-176.322032,-0.120321,-90.000210
C01833=1932.447300,-33.038000,-460.184500,-176.322032,-0.120321,-90.000210
C01834=1931.839200,-33.038000,-460.658400,-176.322032,-0.120321,-90.000210
C01835=1928.033300,-33.038000,-459.392800,-176.322032,-0.120321,-90.000210
C01836=1926.449900,-33.038000,-459.869500,-176.322032,-0.120321,-90.000210
C01837=1922.847200,-33.038000,-459.598400,-176.322032,-0.120321,-90.000210
C01838=1922.331600,-33.038000,-460.286400,-176.322032,-0.120321,-90.000210
C01839=1921.130500,-33.038000,-461.293900,-176.322032,-0.120321,-90.000210
C01840=1917.493100,-33.038000,-460.855700,-176.322032,-0.120321,-90.000210
C01841=1916.540500,-33.038000,-460.962700,-176.322032,-0.120321,-90.000210
C01842=1912.790500,-33.038000,-461.250800,-176.322032,-0.120321,-90.000210
C01843=1911.355900,-33.038000,-460.108000,-176.322032,-0.120321,-90.000210
C01844=1907.391900,-33.038000,-460.981100,-176.322032,-0.120321,-90.000210
C01845=1906.312800,-33.038000,-459.849100,-176.322032,-0.120321,-90.000210
C01846=1903.183400,-33.038000,-459.145100,-176.322032,-0.120321,-90.000210
C01847=1902.901900,-33.038000,-461.310700,-176.322032,-0.120321,-90.000210
C01848=1900.636400,-33.038000,-460.740700,-176.322032,-0.120321,-90.000210
C01849=1897.837200,-33.038000,-460.909400,-176.322032,-0.120321,-90.000210
C01850=1897.597600,-33.038000,-459.241600,-176.322032,-0.120321,-90.000210
C01851=1894.765800,-33.038000,-461.260400,-176.322032,-0.120321,-90.000210
C01852=1892.524100,-33.038000,-459.593400,-176.322032,-0.120321,-90.000210
C01853=1891.819200,-33.038000,-460.231700,-176.322032,-0.120321,-90.000210
C01854=1887.245200,-33.038000,-461.384300,-176.322032,-0.120321,-90.000210
C01855=1886.571600,-33.038000,-459.789700,-176.322032,-0.120321,-90.000210
C01856=1884.738500,-33.038000,-461.008100,-176.322032,-0.120321,-90.000210
C01857=1882.108400,-33.038000,-460.748000,-176.322032,-0.120321,-90.000210
C01858=1880.397600,-33.038000,-459.760200,-176.322032,-0.120321,-90.000210
C01859=1876.965500,-33.038000,-461.214200,-176.322032,-0.120321,-90.000210
C01860=1876.113000,-33.038000,-460.611800,-176.322032,-0.120321,-90.000210
C01861=1872.874700,-33.038000,-460.371600,-176.322032,-0.120321,-90.000210
C01862=1871.807700,-33.038000,-460.314900,-176.322032,-0.120321,-90.000210
C01863=1868.205200,-33.038000,-461.054900,-176.322032,-0.120321,-90.000210
C01864=1866.817300,-33.038000,-458.988800,-176.322032,-0.120321,-90.000210
C01865=1866.123000,-33.038000,-460.006000,-176.322032,-0.120321,-90.000210
C01866=1861.764900,-33.038000,-459.510500,-176.322032,-0.120321,-90.000210
C01867=1861.028000,-33.038000,-460.387900,-176.322032,-0.120321,-90.000210
C01868=1856.776400,-33.038000,-458.848800,-176.322032,-0.120321,-90.000210
C01869=1855.827200,-33.038000,-460.033300,-176.322032,-0.120321,-90.000210
C01870=1851.961700,-33.038000,-459.904400,-176.322032,-0.120321,-90.000210
C01871=1850.635600,-33.038000,-459.546600,-176.322032,-0.120321,-90.000210
C01872=1846.693200,-33.038000,-459.808800,-176.322032,-0.120321,-90.000210
C01873=1846.101900,-33.038000,-459.693200,-176.322032,-0.120321,-90.000210
C01874=1842.005800,-33.038000,-458.706500,-176.322032,-0.120321,-90.000210
C01875=1840.272800,-33.038000,-458.341800,-176.322032,-0.120321,-90.000210
C01876=1836.351700,-33.038000,-458.618600,-176.322032,-0.120321,-90.000210
C01877=1835.877300,-33.038000,-459.666700,-176.322032,-0.120321,-90.000210
C01878=1831.732800,-33.038000,-458.830600,-176.322032,-0.120321,-90.000210
C01879=1827.627900,-33.038000,-458.623500,-176.322032,-0.120321,-90.000210
C01880=1827.146600,-33.038000,-458.251800,-176.322032,-0.120321,-90.000210
C01881=1822.666700,-33.038000,-457.936900,-176.322032,-0.120321,-90.000210
C01882=1821.003600,-33.038000,-458.961100,-176.322032,-0.120321,-90.000210
C01883=1817.553000,-33.038000,-458.342700,-176.322032,-0.120321,-90.000210
C01884=1816.574500,-33.038000,-457.949500,-176.322032,-0.120321,-90.000210
C01885=1812.646800,-33.038000,-458.310900,-176.322032,-0.120321,-90.000210
C01886=1811.813700,-33.038000,-458.144300,-176.322032,-0.120321,-90.000210
C01887=1807.630100,-33.038000,-457.924200,-176.322032,-0.120321,-90.000210
C01888=1806.662700,-33.038000,-457.994800,-176.322032,-0.120321,-90.000210
C01889=1802.325300,-33.038000,-457.304800,-176.322032,-0.120321,-90.000210
C01890=1801.377000,-33.038000,-457.525200,-176.322032,-0.120321,-90.000210
C01891=1797.263700,-83.038000,-456.540200,-176.322032,-0.120321,-90.000210
C01892=1801.377600,-83.038000,-456.423500,-176.322032,-0.120321,-90.000210
C01893=1802.039100,-83.038000,-456.528700,-176.322032,-0.120321,-90.000210
C01894=1806.137700,-83.038000,-456.420600,-176.322032,-0.120321,-90.000210
C01895=1807.517500,-83.038000,-457.040300,-176.322032,-0.120321,-90.000210
C01896=1811.510800,-83.038000,-457.342000,-176.322032,-0.120321,-90.000210
C01897=1812.761400,-83.038000,-456.921400,-176.322032,-0.120321,-90.000210
C01898=1816.633500,-83.038000,-456.944700,-176.322032,-0.120321,-90.000210
C01899=1818.180400,-83.038000,-456.446200,-176.322032,-0.120321,-90.000210
C01900=1821.418400,-83.038000,-457.315100,-176.322032,-0.120321,-90.000210
C01901=1822.147000,-83.038000,-457.631800,-176.322032,-0.120321,-90.000210
C01902=1825.940600,-83.038000,-457.200100,-176.322032,-0.120321,-90.000210
C01903=1827.184000,-83.038000,-456.413500,-176.322032,-0.120321,-90.000210
C01904=1831.431900,-83.038000,-456.952100,-176.322032,-0.120321,-90.000210
C01905=1832.943800,-83.038000,-457.695100,-176.322032,-0.120321,-90.000210
C01906=1836.336500,-83.038000,-456.649600,-176.322032,-0.120321,-90.000210
C01907=1837.917700,-83.038000,-456.259000,-176.322032,-0.120321,-90.000210
C01908=1841.653600,-83.038000,-456.294100,-176.322032,-0.120321,-90.000210
C01909=1842.500500,-83.038000,-457.453300,-176.322032,-0.120321,-90.000210
C01910=1846.655000,-83.038000,-456.158800,-176.322032,-0.120321,-90.000210
C01911=1847.914100,-83.038000,-456.971400,-176.322032,-0.120321,-90.000210
C01912=1850.886400,-83.038000,-457.947500,-176.322032,-0.120321,-90.000210
C01913=1851.924300,-83.038000,-456.455900,-176.322032,-0.120321,-90.000210
C01914=1853.746500,-83.038000,-455.909000,-176.322032,-0.120321,-90.000210
C01915=1856.801000,-83.038000,-456.540700,-176.322032,-0.120321,-90.000210
C01916=1857.226900,-83.038000,-457.572000,-176.322032,-0.120321,-90.000210
C01917=1861.661500,-83.038000,-457.096300,-176.322032,-0.120321,-90.000210
C01918=1862.298300,-83.038000,-456.125500,-176.322032,-0.120321,-90.000210
C01919=1866.796100,-83.038000,-456.521100,-176.322032,-0.120321,-90.000210
C01920=1868.461700,-83.038000,-457.691500,-176.322032,-0.120321,-90.000210
C01921=1871.614500,-83.038000,-458.087100,-176.322032,-0.120321,-90.000210
C01922=1872.861100,-83.038000,-457.346300,-176.322032,-0.120321,-90.000210
C01923=1876.567400,-83.038000,-457.369000,-176.322032,-0.120321,-90.000210
C01924=1877.660500,-83.038000,-456.269800,-176.322032,-0.120321,-90.000210
C01925=1881.048400,-83.038000,-455.876700,-176.322032,-0.120321,-90.000210
C01926=1882.363100,-83.038000,-456.205000,-176.322032,-0.120321,-90.000210
C01927=1885.185000,-83.038000,-458.324900,-176.322032,-0.120321,-90.000210
C01928=1886.931500,-83.038000,-457.616100,-176.322032,-0.120321,-90.000210
C01929=1891.295700,-83.038000,-456.342800,-176.322032,-0.120321,-90.000210
C01930=1892.497100,-83.038000,-456.878000,-176.322032,-0.120321,-90.000210
C01931=1895.995100,-83.038000,-455.878400,-176.322032,-0.120321,-90.000210
C01932=1897.742400,-83.038000,-457.729200,-176.322032,-0.120321,-90.000210
C01933=1901.249700,-83.038000,-458.023200,-176.322032,-0.120321,-90.000210
C01934=1902.218000,-83.038000,-457.070400,-176.322032,-0.120321,-90.000210
C01935=1904.345200,-83.038000,-456.433500,-176.322032,-0.120321,-90.000210
C01936=1906.979400,-83.038000,-457.295900,-176.322032,-0.120321,-90.000210
C01937=1909.333600,-83.038000,-458.869800,-176.322032,-0.120321,-90.000210
C01938=1911.531500,-83.038000,-456.868200,-176.322032,-0.120321,-90.000210
C01939=1912.668800,-83.038000,-456.031500,-176.322032,-0.120321,-90.000210
C01940=1916.918700,-83.038000,-458.426000,-176.322032,-0.120321,-90.000210
C01941=1917.701900,-83.038000,-457.524600,-176.322032,-0.120321,-90.000210
C01942=1922.078500,-83.038000,-458.064100,-176.322032,-0.120321,-90.000210
C01943=1922.918000,-83.038000,-457.294700,-176.322032,-0.120321,-90.000210
C01944=1926.700100,-83.038000,-459.205300,-176.322032,-0.120321,-90.000210
C01945=1927.250900,-83.038000,-457.182000,-176.322032,-0.120321,-90.000210
C01946=1931.982400,-83.038000,-456.069000,-176.322032,-0.120321,-90.000210
C01947=1932.147700,-83.038000,-457.389500,-176.322032,-0.120321,-90.000210
C01948=1936.037800,-83.038000,-455.685800,-176.322032,-0.120321,-90.000210
C01949=1937.405100,-83.038000,-458.998100,-176.322032,-0.120321,-90.000210
C01950=1940.796800,-83.038000,-456.815200,-176.322032,-0.120321,-90.000210
C01951=1942.395200,-83.038000,-457.390500,-176.322032,-0.120321,-90.000210
C01952=1944.845500,-83.038000,-458.958400,-176.322032,-0.120321,-90.000210
C01953=1946.875900,-83.038000,-456.942200,-176.322032,-0.120321,-90.000210
C01954=1950.220400,-83.038000,-456.395300,-176.322032,-0.120321,-90.000210
C01955=1951.914900,-83.038000,-457.328000,-176.322032,-0.120321,-90.000210
C01956=1955.423500,-83.038000,-456.371300,-176.322032,-0.120321,-90.000210
C01957=1956.995800,-83.038000,-458.267900,-176.322032,-0.120321,-90.000210
C01958=1959.602900,-83.038000,-456.606400,-176.322032,-0.120321,-90.000210
C01959=1961.519200,-83.038000,-458.740100,-176.322032,-0.120321,-90.000210
C01960=1965.354500,-83.038000,-457.213900,-176.322032,-0.120321,-90.000210
C01961=1966.905300,-83.038000,-455.640300,-176.322032,-0.120321,-90.000210
C01962=1971.058500,-83.038000,-457.727600,-176.322032,-0.120321,-90.000210
C01963=1972.264700,-83.038000,-456.054500,-176.322032,-0.120321,-90.000210
C01964=1974.115900,-83.038000,-455.778900,-176.322032,-0.120321,-90.000210
C01965=1976.905200,-83.038000,-457.645300,-176.322032,-0.120321,-90.000210
C01966=1977.676300,-83.038000,-458.975900,-176.322032,-0.120321,-90.000210
C01967=1981.825400,-83.038000,-457.787200,-176.322032,-0.120321,-90.000210
C01968=1983.003600,-83.038000,-456.479500,-176.322032,-0.120321,-90.000210
C01969=1986.886100,-83.038000,-458.067200,-176.322032,-0.120321,-90.000210
C01970=1989.294000,-83.038000,-455.376600,-176.322032,-0.120321,-90.000210
C01971=1992.332000,-83.038000,-457.244500,-176.322032,-0.120321,-90.000210
C01972=1994.263900,-83.038000,-458.489200,-176.322032,-0.120321,-90.000210
C01973=1996.329700,-83.038000,-458.739300,-176.322032,-0.120321,-90.000210
C01974=1997.462100,-83.038000,-458.441800,-176.322032,-0.120321,-90.000210
C01975=2001.519800,-83.038000,-456.471900,-176.322032,-0.120321,-90.000210
C01976=2002.039100,-83.038000,-458.226600,-176.322032,-0.120321,-90.000210
C01977=2006.365200,-83.038000,-457.899400,-176.322032,-0.120321,-90.000210
C01978=2007.611500,-83.038000,-456.940000,-176.322032,-0.120321,-90.000210
C01979=2011.393600,-83.038000,-457.792900,-176.322032,-0.120321,-90.000210
C01980=2012.219700,-83.038000,-456.288200,-176.322032,-0.120321,-90.000210
C01981=2015.812100,-83.038000,-458.440800,-176.322032,-0.120321,-90.000210
C01982=2017.030100,-83.038000,-456.217900,-176.322032,-0.120321,-90.000210
C01983=2021.279300,-83.038000,-458.175600,-176.322032,-0.120321,-90.000210
C01984=2022.237300,-83.038000,-456.596800,-176.322032,-0.120321,-90.000210
C01985=2026.020400,-83.038000,-457.311200,-176.322032,-0.120321,-90.000210
C01986=2026.631900,-83.038000,-456.498800,-176.322032,-0.120321,-90.000210
C01987=2030.724300,-83.038000,-456.286000,-176.322032,-0.120321,-90.000210
C01988=2031.361900,-83.038000,-458.301200,-176.322032,-0.120321,-90.000210
C01989=2035.954200,-83.038000,-458.269700,-176.322032,-0.120321,-90.000210
C01990=2037.154700,-83.038000,-456.120400,-176.322032,-0.120321,-90.000210
C01991=2038.215800,-83.038000,-455.719800,-176.322032,-0.120321,-90.000210
C01992=2042.068600,-83.038000,-457.753500,-176.322032,-0.120321,-90.000210
C01993=2043.184400,-83.038000,-456.910400,-176.322032,-0.120321,-90.000210
C01994=2046.139200,-83.038000,-458.371800,-176.322032,-0.120321,-90.000210
C01995=2046.949300,-83.038000,-456.269600,-176.322032,-0.120321,-90.000210
C01996=2051.275500,-83.038000,-458.065400,-176.322032,-0.120321,-90.000210
C01997=2052.389700,-83.038000,-458.406500,-176.322032,-0.120321,-90.000210
C01998=2056.771500,-83.038000,-457.622900,-176.322032,-0.120321,-90.000210
C01999=2057.436900,-83.038000,-456.230700,-176.322032,-0.120321,-90.000210
C02000=2061.046500,-83.038000,-458.471100,-176.322032,-0.120321,-90.000210
C02001=2062.307600,-83.038000,-458.250100,-176.322032,-0.120321,-90.000210
C02002=2066.484400,-83.038000,-456.692500,-176.322032,-0.120321,-90.000210
C02003=2067.746400,-83.038000,-456.025700,-176.322032,-0.120321,-90.000210
C02004=2069.633900,-83.038000,-456.869800,-176.322032,-0.120321,-90.000210
C02005=2071.554400,-83.038000,-455.892900,-176.322032,-0.120321,-90.000210
C02006=2072.633200,-83.038000,-457.582900,-176.322032,-0.120321,-90.000210
C02007=2076.333700,-83.038000,-457.344400,-176.322032,-0.120321,-90.000210
C02008=2077.954900,-83.038000,-457.572800,-176.322032,-0.120321,-90.000210
C02009=2081.587400,-83.038000,-458.305800,-176.322032,-0.120321,-90.000210
C02010=2082.795300,-83.038000,-457.300800,-176.322032,-0.120321,-90.000210
C02011=2086.722900,-83.038000,-457.167600,-176.322032,-0.120321,-90.000210
C02012=2088.396100,-83.038000,-455.635400,-176.322032,-0.120321,-90.000210
C02013=2091.369400,-83.038000,-457.029000,-176.322032,-0.120321,-90.000210
C02014=2092.142400,-83.038000,-456.409600,-176.322032,-0.120321,-90.000210
C02015=2096.407500,-83.038000,-457.112600,-176.322032,-0.120321,-90.000210
C02016=2098.017100,-83.038000,-456.330700,-176.322032,-0.120321,-90.000210
C02017=2101.502400,-83.038000,-456.888600,-176.322032,-0.120321,-90.000210
C02018=2102.273900,-83.038000,-457.221300,-176.322032,-0.120321,-90.000210
C02019=2106.143100,-83.038000,-455.631300,-176.322032,-0.120321,-90.000210
C02020=2106.749400,-83.038000,-456.158000,-176.322032,-0.120321,-90.000210
C02021=2109.791900,-83.038000,-455.916200,-176.322032,-0.120321,-90.000210
C02022=2112.245200,-83.038000,-457.240800,-176.322032,-0.120321,-90.000210
C02023=2113.650000,-83.038000,-456.224800,-176.322032,-0.120321,-90.000210
C02024=2116.592900,-83.038000,-457.485200,-176.322032,-0.120321,-90.000210
C02025=2118.171700,-83.038000,-457.734300,-176.322032,-0.120321,-90.000210
C02026=2121.489400,-83.038000,-455.713700,-176.322032,-0.120321,-90.000210
C02027=2123.002800,-83.038000,-456.620500,-176.322032,-0.120321,-90.000210
C02028=2126.272600,-83.038000,-456.458500,-176.322032,-0.120321,-90.000210
C02029=2127.021400,-83.038000,-456.241800,-176.322032,-0.120321,-90.000210
C02030=2130.380500,-83.038000,-455.975500,-176.322032,-0.120321,-90.000210
C02031=2131.517900,-83.038000,-456.490200,-176.322032,-0.120321,-90.000210
C02032=2133.000400,-83.038000,-457.288100,-176.322032,-0.120321,-90.000210
C02033=2136.544700,-83.038000,-456.314300,-176.322032,-0.120321,-90.000210
C02034=2137.561500,-83.038000,-456.582300,-176.322032,-0.120321,-90.000210
C02035=2140.485200,-83.038000,-456.953300,-176.322032,-0.120321,-90.000210
C02036=2142.027500,-83.038000,-455.560600,-176.322032,-0.120321,-90.000210
C02037=2143.171400,-83.038000,-455.414800,-176.322032,-0.120321,-90.000210
C02038=2146.645500,-83.038000,-455.859300,-176.322032,-0.120321,-90.000210
C02039=2147.458000,-83.038000,-455.621500,-176.322032,-0.120321,-90.000210
C02040=2151.204600,-83.038000,-456.511100,-176.322032,-0.120321,-90.000210
C02041=2152.489100,-83.038000,-455.289500,-176.322032,-0.120321,-90.000210
C02042=2156.219900,-83.038000,-454.624000,-176.322032,-0.120321,-90.000210
C02043=2157.348100,-83.038000,-456.405500,-176.322032,-0.120321,-90.000210
C02044=2160.882400,-83.038000,-455.794700,-176.322032,-0.120321,-90.000210
C02045=2161.954200,-83.038000,-456.106900,-176.322032,-0.120321,-90.000210
C02046=2164.616700,-83.038000,-456.092100,-176.322032,-0.120321,-90.000210
C02047=2167.074500,-83.038000,-455.772800,-176.322032,-0.120321,-90.000210
C02048=2168.424400,-83.038000,-455.258200,-176.322032,-0.120321,-90.000210
C02049=2171.813600,-83.038000,-455.571700,-176.322032,-0.120321,-90.000210
C02050=2173.005300,-83.038000,-455.054600,-176.322032,-0.120321,-90.000210
C02051=2176.119100,-83.038000,-455.289600,-176.322032,-0.120321,-90.000210
C02052=2177.224700,-83.038000,-454.727600,-176.322032,-0.120321,-90.000210
C02053=2181.520500,-83.038000,-454.439800,-176.322032,-0.120321,-90.000210
C02054=2182.514000,-83.038000,-455.350200,-176.322032,-0.120321,-90.000210
C02055=2185.997400,-83.038000,-454.048100,-176.322032,-0.120321,-90.000210
C02056=2187.456900,-83.038000,-453.822700,-176.322032,-0.120321,-90.000210
C02057=2187.373800,-133.038000,-453.058600,-176.322032,-0.120321,-90.000210
C02058=2186.173000,-133.038000,-452.904400,-176.322032,-0.120321,-90.000210
C02059=2181.970900,-133.038000,-453.572100,-176.322032,-0.120321,-90.000210
C02060=2181.086000,-133.038000,-452.259200,-176.322032,-0.120321,-90.000210
C02061=2177.642900,-133.038000,-452.841500,-176.322032,-0.120321,-90.000210
C02062=2176.178200,-133.038000,-454.289400,-176.322032,-0.120321,-90.000210
C02063=2172.448000,-133.038000,-453.722100,-176.322032,-0.120321,-90.000210
C02064=2171.093000,-133.038000,-454.267900,-176.322032,-0.120321,-90.000210
C02065=2167.273800,-133.038000,-452.746200,-176.322032,-0.120321,-90.000210
C02066=2166.588800,-133.038000,-454.231300,-176.322032,-0.120321,-90.000210
C02067=2162.219200,-133.038000,-453.252000,-176.322032,-0.120321,-90.000210
C02068=2161.345900,-133.038000,-454.239100,-176.322032,-0.120321,-90.000210
C02069=2157.321500,-133.038000,-453.888100,-176.322032,-0.120321,-90.000210
C02070=2156.881400,-133.038000,-454.395000,-176.322032,-0.120321,-90.000210
C02071=2152.391800,-133.038000,-453.025200,-176.322032,-0.120321,-90.000210
C02072=2151.094200,-133.038000,-453.392500,-176.322032,-0.120321,-90.000210
C02073=2147.436600,-133.038000,-454.712900,-176.322032,-0.120321,-90.000210
C02074=2146.105500,-133.038000,-452.489700,-176.322032,-0.120321,-90.000210
C02075=2142.728200,-133.038000,-453.775300,-176.322032,-0.120321,-90.000210
C02076=2141.248700,-133.038000,-452.540700,-176.322032,-0.120321,-90.000210
C02077=2137.222500,-133.038000,-454.428400,-176.322032,-0.120321,-90.000210
C02078=2135.926800,-133.038000,-452.055400,-176.322032,-0.120321,-90.000210
C02079=2132.036600,-133.038000,-454.675800,-176.322032,-0.120321,-90.000210
C02080=2131.072200,-133.038000,-452.371800,-176.322032,-0.120321,-90.000210
C02081=2127.231500,-133.038000,-454.577500,-176.322032,-0.120321,-90.000210
C02082=2126.719800,-133.038000,-455.046800,-176.322032,-0.120321,-90.000210
C02083=2122.286700,-133.038000,-454.057800,-176.322032,-0.120321,-90.000210
C02084=2120.565600,-133.038000,-454.499500,-176.322032,-0.120321,-90.000210
C02085=2117.277500,-133.038000,-451.748900,-176.322032,-0.120321,-90.000210
C02086=2115.704300,-133.038000,-454.725800,-176.322032,-0.120321,-90.000210
C02087=2112.314000,-133.038000,-455.309700,-176.322032,-0.120321,-90.000210
C02088=2111.374800,-133.038000,-454.773000,-176.322032,-0.120321,-90.000210
C02089=2106.960300,-133.038000,-454.636700,-176.322032,-0.120321,-90.000210
C02090=2106.224500,-133.038000,-451.947200,-176.322032,-0.120321,-90.000210
C02091=2102.475600,-133.038000,-454.889200,-176.322032,-0.120321,-90.000210
C02092=2101.684300,-133.038000,-454.016100,-176.322032,-0.120321,-90.000210
C02093=2097.394700,-133.038000,-453.504300,-176.322032,-0.120321,-90.000210
C02094=2096.126000,-133.038000,-453.711500,-176.322032,-0.120321,-90.000210
C02095=2092.164600,-133.038000,-454.984800,-176.322032,-0.120321,-90.000210
C02096=2091.068400,-133.038000,-453.204200,-176.322032,-0.120321,-90.000210
C02097=2087.539000,-133.038000,-454.995900,-176.322032,-0.120321,-90.000210
C02098=2086.319500,-133.038000,-453.344600,-176.322032,-0.120321,-90.000210
C02099=2082.211700,-133.038000,-452.721300,-176.322032,-0.120321,-90.000210
C02100=2081.793900,-133.038000,-455.285200,-176.322032,-0.120321,-90.000210
C02101=2076.871800,-133.038000,-455.786500,-176.322032,-0.120321,-90.000210
C02102=2075.480800,-133.038000,-454.697700,-176.322032,-0.120321,-90.000210
C02103=2071.132500,-133.038000,-452.233100,-176.322032,-0.120321,-90.000210
C02104=2068.360600,-133.038000,-453.353800,-176.322032,-0.120321,-90.000210
C02105=2066.886600,-133.038000,-454.523600,-176.322032,-0.120321,-90.000210
C02106=2063.419300,-133.038000,-454.885100,-176.322032,-0.120321,-90.000210
C02107=2061.568500,-133.038000,-455.500200,-176.322032,-0.120321,-90.000210
C02108=2057.624800,-133.038000,-455.500900,-176.322032,-0.120321,-90.000210
C02109=2057.004000,-133.038000,-454.887100,-176.322032,-0.120321,-90.000210
C02110=2053.191200,-133.038000,-453.109900,-176.322032,-0.120321,-90.000210
C02111=2051.756600,-133.038000,-455.206700,-176.322032,-0.120321,-90.000210
C02112=2048.678100,-133.038000,-455.166800,-176.322032,-0.120321,-90.000210
C02113=2047.198200,-133.038000,-451.334300,-176.322032,-0.120321,-90.000210
C02114=2043.365000,-133.038000,-453.901600,-176.322032,-0.120321,-90.000210
C02115=2041.721000,-133.038000,-453.658900,-176.322032,-0.120321,-90.000210
C02116=2037.967200,-133.038000,-452.938200,-176.322032,-0.120321,-90.000210
C02117=2036.885000,-133.038000,-452.406200,-176.322032,-0.120321,-90.000210
C02118=2032.344200,-133.038000,-453.994900,-176.322032,-0.120321,-90.000210
C02119=2031.784900,-133.038000,-453.270900,-176.322032,-0.120321,-90.000210
C02120=2028.013600,-133.038000,-454.885300,-176.322032,-0.120321,-90.000210
C02121=2026.752200,-133.038000,-451.706600,-176.322032,-0.120321,-90.000210
C02122=2022.750300,-133.038000,-452.672800,-176.322032,-0.120321,-90.000210
C02123=2021.130800,-133.038000,-454.197800,-176.322032,-0.120321,-90.000210
C02124=2018.221600,-133.038000,-456.075300,-176.322032,-0.120321,-90.000210
C02125=2016.328300,-133.038000,-454.195800,-176.322032,-0.120321,-90.000210
C02126=2012.311500,-133.038000,-453.970100,-176.322032,-0.120321,-90.000210
C02127=2011.246900,-133.038000,-455.091600,-176.322032,-0.120321,-90.000210
C02128=2007.556100,-133.038000,-454.730500,-176.322032,-0.120321,-90.000210
C02129=2006.472900,-133.038000,-455.380500,-176.322032,-0.120321,-90.000210
C02130=2001.970100,-133.038000,-452.315200,-176.322032,-0.120321,-90.000210
C02131=2000.601800,-133.038000,-455.368300,-176.322032,-0.120321,-90.000210
C02132=1997.453700,-133.038000,-454.754800,-176.322032,-0.120321,-90.000210
C02133=1996.489900,-133.038000,-453.154200,-176.322032,-0.120321,-90.000210
C02134=1992.029300,-133.038000,-454.096800,-176.322032,-0.120321,-90.000210
C02135=1991.548200,-133.038000,-453.439600,-176.322032,-0.120321,-90.000210
C02136=1986.869000,-133.038000,-453.776100,-176.322032,-0.120321,-90.000210
C02137=1985.820000,-133.038000,-453.951500,-176.322032,-0.120321,-90.000210
C02138=1982.350200,-133.038000,-453.250800,-176.322032,-0.120321,-90.000210
C02139=1981.268400,-133.038000,-454.339200,-176.322032,-0.120321,-90.000210
C02140=1977.068200,-133.038000,-455.258900,-176.322032,-0.120321,-90.000210
C02141=1976.165200,-133.038000,-454.760800,-176.322032,-0.120321,-90.000210
C02142=1972.187500,-133.038000,-453.934700,-176.322032,-0.120321,-90.000210
C02143=1971.166300,-133.038000,-454.891400,-176.322032,-0.120321,-90.000210
C02144=1967.473700,-133.038000,-454.101600,-176.322032,-0.120321,-90.000210
C02145=1966.060900,-133.038000,-455.392900,-176.322032,-0.120321,-90.000210
C02146=1961.675900,-133.038000,-454.814300,-176.322032,-0.120321,-90.000210
C02147=1961.012700,-133.038000,-452.894300,-176.322032,-0.120321,-90.000210
C02148=1956.743800,-133.038000,-453.982200,-176.322032,-0.120321,-90.000210
C02149=1956.343300,-133.038000,-454.968300,-176.322032,-0.120321,-90.000210
C02150=1952.013600,-133.038000,-454.486200,-176.322032,-0.120321,-90.000210
C02151=1951.398800,-133.038000,-454.244500,-176.322032,-0.120321,-90.000210
C02152=1947.484700,-133.038000,-455.723300,-176.322032,-0.120321,-90.000210
C02153=1946.181200,-133.038000,-453.128600,-176.322032,-0.120321,-90.000210
C02154=1942.188600,-133.038000,-455.373800,-176.322032,-0.120321,-90.000210
C02155=1941.485900,-133.038000,-456.084500,-176.322032,-0.120321,-90.000210
C02156=1937.171800,-133.038000,-452.942700,-176.322032,-0.120321,-90.000210
C02157=1936.777700,-133.038000,-454.336100,-176.322032,-0.120321,-90.000210
C02158=1932.595400,-133.038000,-454.888800,-176.322032,-0.120321,-90.000210
C02159=1931.693900,-133.038000,-455.408800,-176.322032,-0.120321,-90.000210
C02160=1927.858800,-133.038000,-454.821700,-176.322032,-0.120321,-90.000210
C02161=1926.659200,-133.038000,-452.831500,-176.322032,-0.120321,-90.000210
C02162=1922.429200,-133.038000,-455.521300,-176.322032,-0.120321,-90.000210
C02163=1921.791500,-133.038000,-455.397000,-176.322032,-0.120321,-90.000210
C02164=1918.851000,-133.038000,-454.800000,-176.322032,-0.120321,-90.000210
C02165=1917.010700,-133.038000,-452.245200,-176.322032,-0.120321,-90.000210
C02166=1914.019500,-133.038000,-455.955100,-176.322032,-0.120321,-90.000210
C02167=1912.257600,-133.038000,-454.967400,-176.322032,-0.120321,-90.000210
C02168=1910.541300,-133.038000,-455.157900,-176.322032,-0.120321,-90.000210
C02169=1907.346700,-133.038000,-452.907900,-176.322032,-0.120321,-90.000210
C02170=1905.944000,-133.038000,-455.678800,-176.322032,-0.120321,-90.000210
C02171=1902.008600,-133.038000,-455.767400,-176.322032,-0.120321,-90.000210
C02172=1901.152900,-133.038000,-455.565200,-176.322032,-0.120321,-90.000210
C02173=1897.458300,-133.038000,-453.701900,-176.322032,-0.120321,-90.000210
C02174=1896.226900,-133.038000,-455.974900,-176.322032,-0.120321,-90.000210
C02175=1892.459100,-133.038000,-454.184900,-176.322032,-0.120321,-90.000210
C02176=1891.454300,-133.038000,-455.045000,-176.322032,-0.120321,-90.000210
C02177=1887.301200,-133.038000,-455.639500,-176.322032,-0.120321,-90.000210
C02178=1887.094000,-133.038000,-454.789800,-176.322032,-0.120321,-90.000210
C02179=1881.707500,-133.038000,-454.831600,-176.322032,-0.120321,-90.000210
C02180=1880.935000,-133.038000,-454.177700,-176.322032,-0.120321,-90.000210
C02181=1877.465500,-133.038000,-455.617600,-176.322032,-0.120321,-90.000210
C02182=1876.452400,-133.038000,-453.948400,-176.322032,-0.120321,-90.000210
C02183=1872.152900,-133.038000,-453.644800,-176.322032,-0.120321,-90.000210
C02184=1871.251700,-133.038000,-454.462300,-176.322032,-0.120321,-90.000210
C02185=1867.034600,-133.038000,-455.314900,-176.322032,-0.120321,-90.000210
C02186=1866.363300,-133.038000,-454.623500,-176.322032,-0.120321,-90.000210
C02187=1861.762500,-133.038000,-454.870800,-176.322032,-0.120321,-90.000210
C02188=1860.357000,-133.038000,-454.604400,-176.322032,-0.120321,-90.000210
C02189=1856.822700,-133.038000,-454.995400,-176.322032,-0.120321,-90.000210
C02190=1855.793100,-133.038000,-453.836500,-176.322032,-0.120321,-90.000210
C02191=1852.369400,-133.038000,-454.282900,-176.322032,-0.120321,-90.000210
C02192=1851.706700,-133.038000,-454.546100,-176.322032,-0.120321,-90.000210
C02193=1847.013900,-133.038000,-454.673200,-176.322032,-0.120321,-90.000210
C02194=1846.392900,-133.038000,-456.104600,-176.322032,-0.120321,-90.000210
C02195=1842.853400,-133.038000,-454.701400,-176.322032,-0.120321,-90.000210
C02196=1841.764100,-133.038000,-455.566400,-176.322032,-0.120321,-90.000210
C02197=1837.893700,-133.038000,-456.110000,-176.322032,-0.120321,-90.000210
C02198=1836.646400,-133.038000,-454.832900,-176.322032,-0.120321,-90.000210
C02199=1834.854100,-133.038000,-455.757000,-176.322032,-0.120321,-90.000210
C02200=1831.290000,-133.038000,-454.943100,-176.322032,-0.120321,-90.000210
C02201=1827.575100,-133.038000,-455.770900,-176.322032,-0.120321,-90.000210
C02202=1826.678600,-133.038000,-455.706400,-176.322032,-0.120321,-90.000210
C02203=1825.333700,-133.038000,-455.274200,-176.322032,-0.120321,-90.000210
C02204=1822.107100,-133.038000,-455.697600,-176.322032,-0.120321,-90.000210
C02205=1821.345000,-133.038000,-456.237900,-176.322032,-0.120321,-90.000210
C02206=1819.592600,-133.038000,-456.016000,-176.322032,-0.120321,-90.000210
C02207=1817.152700,-133.038000,-456.207500,-176.322032,-0.120321,-90.000210
C02208=1815.752400,-133.038000,-456.162400,-176.322032,-0.120321,-90.000210
C02209=1812.473500,-133.038000,-455.878000,-176.322032,-0.120321,-90.000210
C02210=1811.262800,-133.038000,-455.512600,-176.322032,-0.120321,-90.000210
C02211=1807.875800,-133.038000,-456.284700,-176.322032,-0.120321,-90.000210
C02212=1807.109300,-133.038000,-456.069700,-176.322032,-0.120321,-90.000210
C02213=1805.572300,-133.038000,-455.935000,-176.322032,-0.120321,-90.000210
C02214=1802.605100,-133.038000,-455.813800,-176.322032,-0.120321,-90.000210
C02215=1801.855500,-133.038000,-456.078200,-176.322032,-0.120321,-90.000210
C02216=1800.000800,-133.038000,-456.024600,-176.322032,-0.120321,-90.000210
C02217=1796.212400,-133.038000,-456.323000,-176.322032,-0.120321,-90.000210
C02218=1811.635000,221.108300,-503.720300,90.647653,-0.183346,-0.000000
C02219=2127.176000,221.135000,-503.720300,90.647653,-0.183346,-0.000000
C02220=2158.549300,221.162700,-503.720300,90.647653,-0.183346,-0.000000
C02221=1815.760400,221.193100,-503.720300,90.647653,-0.183346,-0.000000
C02222=1821.263900,221.224800,-503.720300,90.647653,-0.183346,-0.000000
C02223=1812.312200,221.239900,-503.720300,90.647653,-0.183346,-0.000000
C02224=1809.093700,221.252000,-503.720300,90.647653,-0.183346,-0.000000
C02225=1831.237900,221.270100,-503.720300,90.647653,-0.183346,-0.000000
C02226=1825.910000,221.290400,-503.720300,90.647653,-0.183346,-0.000000
C02227=1834.967300,221.302200,-503.720300,90.647653,-0.183346,-0.000000
C02228=1839.702600,221.325900,-503.720300,90.647653,-0.183346,-0.000000
C02229=1835.410300,221.337300,-503.720300,90.647653,-0.183346,-0.000000
C02230=2118.838500,221.344100,-503.720300,90.647653,-0.183346,-0.000000
C02231=2151.568300,221.348800,-503.720300,90.647653,-0.183346,-0.000000
C02232=2174.762900,221.357600,-503.720300,90.647653,-0.183346,-0.000000
C02233=1808.009800,221.388700,-503.720300,90.647653,-0.183346,-0.000000
C02234=2144.201400,221.400900,-503.720300,90.647653,-0.183346,-0.000000
C02235=1798.112100,221.410000,-503.720300,90.647653,-0.183346,-0.000000
C02236=1837.822200,221.419800,-503.720300,90.647653,-0.183346,-0.000000
C02237=2112.433200,221.443100,-503.720300,90.647653,-0.183346,-0.000000
C02238=2136.213500,221.451500,-503.720300,90.647653,-0.183346,-0.000000
C02239=2089.573900,221.466700,-503.720300,90.647653,-0.183346,-0.000000
C02240=1866.266000,221.478900,-503.720300,90.647653,-0.183346,-0.000000
C02241=2119.282900,221.493800,-503.720300,90.647653,-0.183346,-0.000000
C02242=1857.771200,221.511800,-503.720300,90.647653,-0.183346,-0.000000
C02243=2166.291900,221.526500,-503.720300,90.647653,-0.183346,-0.000000
C02244=1850.974600,221.541100,-503.720300,90.647653,-0.183346,-0.000000
C02245=2143.673000,221.556300,-503.720300,90.647653,-0.183346,-0.000000
C02246=1828.630300,221.583500,-503.720300,90.647653,-0.183346,-0.000000
C02247=1860.958700,221.587300,-503.720300,90.647653,-0.183346,-0.000000
C02248=2184.435100,221.597500,-503.720300,90.647653,-0.183346,-0.000000
C02249=2090.804900,221.609300,-503.720300,90.647653,-0.183346,-0.000000
C02250=1817.450100,221.621800,-503.720300,90.647653,-0.183346,-0.000000
C02251=2128.070000,221.637700,-503.720300,90.647653,-0.183346,-0.000000
C02252=2189.176300,221.647500,-503.720300,90.647653,-0.183346,-0.000000
C02253=2117.034000,221.655300,-503.720300,90.647653,-0.183346,-0.000000
C02254=2108.809800,221.660300,-503.720300,90.647653,-0.183346,-0.000000
C02255=2089.962200,221.676200,-503.720300,90.647653,-0.183346,-0.000000
C02256=2113.622500,221.682600,-503.720300,90.647653,-0.183346,-0.000000
C02257=2125.630600,221.687300,-503.720300,90.647653,-0.183346,-0.000000
C02258=2088.737700,221.698800,-503.720300,90.647653,-0.183346,-0.000000
C02259=1865.593300,221.709000,-503.720300,90.647653,-0.183346,-0.000000
C02260=2127.249600,221.720500,-503.720300,90.647653,-0.183346,-0.000000
C02261=2081.446100,221.733300,-503.720300,90.647653,-0.183346,-0.000000
C02262=2078.914800,221.740800,-503.720300,90.647653,-0.183346,-0.000000
C02263=1876.021100,221.753900,-503.720300,90.647653,-0.183346,-0.000000
C02264=1875.515000,221.766700,-503.720300,90.647653,-0.183346,-0.000000
C02265=2183.148600,221.795100,-503.720300,90.647653,-0.183346,-0.000000
C02266=2072.022500,221.806300,-503.720300,90.647653,-0.183346,-0.000000
C02267=2079.695800,221.820800,-503.720300,90.647653,-0.183346,-0.000000
C02268=1887.088100,221.832300,-503.720300,90.647653,-0.183346,-0.000000
C02269=2188.540200,221.850500,-503.720300,90.647653,-0.183346,-0.000000
C02270=2075.988300,221.856300,-503.720300,90.647653,-0.183346,-0.000000
C02271=2063.126900,221.863400,-503.720300,90.647653,-0.183346,-0.000000
C02272=1880.005300,221.883000,-503.720300,90.647653,-0.183346,-0.000000
C02273=2072.176800,221.892200,-503.720300,90.647653,-0.183346,-0.000000
C02274=2142.155500,221.923200,-503.720300,90.647653,-0.183346,-0.000000
C02275=2163.272300,221.942100,-503.720300,90.647653,-0.183346,-0.000000
C02276=2043.282500,221.953200,-503.720300,90.647653,-0.183346,-0.000000
C02277=2143.086100,221.981600,-503.720300,90.647653,-0.183346,-0.000000
C02278=2151.779800,221.997200,-503.720300,90.647653,-0.183346,-0.000000
C02279=1889.947900,222.011300,-503.720300,90.647653,-0.183346,-0.000000
C02280=2187.503800,222.024700,-503.720300,90.647653,-0.183346,-0.000000
C02281=1997.220300,222.037400,-503.720300,90.647653,-0.183346,-0.000000
C02282=1908.585700,222.055600,-503.720300,90.647653,-0.183346,-0.000000
C02283=1902.103800,222.075200,-503.720300,90.647653,-0.183346,-0.000000
C02284=1894.253500,222.092100,-503.720300,90.647653,-0.183346,-0.000000
C02285=2087.902000,222.095600,-503.720300,90.647653,-0.183346,-0.000000
C02286=1918.899200,222.119100,-503.720300,90.647653,-0.183346,-0.000000
C02287=1997.786400,222.136500,-503.720300,90.647653,-0.183346,-0.000000
C02288=1996.583100,222.154600,-503.720300,90.647653,-0.183346,-0.000000
C02289=1985.344900,222.169500,-503.720300,90.647653,-0.183346,-0.000000
C02290=1910.038100,222.180600,-503.720300,90.647653,-0.183346,-0.000000
C02291=2048.549000,222.196100,-503.720300,90.647653,-0.183346,-0.000000
C02292=2035.591900,222.207300,-503.720300,90.647653,-0.183346,-0.000000
C02293=2032.094500,222.238400,-503.720300,90.647653,-0.183346,-0.000000
C02294=1901.470500,222.247800,-503.720300,90.647653,-0.183346,-0.000000
C02295=1911.640600,222.265500,-503.720300,90.647653,-0.183346,-0.000000
C02296=2025.335900,222.272500,-503.720300,90.647653,-0.183346,-0.000000
C02297=1897.938300,222.297800,-503.720300,90.647653,-0.183346,-0.000000
C02298=2028.686800,222.312700,-503.720300,90.647653,-0.183346,-0.000000
C02299=1901.595600,222.321100,-503.720300,90.647653,-0.183346,-0.000000
C02300=1927.085400,222.331600,-503.720300,90.647653,-0.183346,-0.000000
C02301=2002.627400,222.354900,-503.720300,90.647653,-0.183346,-0.000000
C02302=1981.632500,222.370800,-503.720300,90.647653,-0.183346,-0.000000
C02303=2008.400500,222.382000,-503.720300,90.647653,-0.183346,-0.000000
C02304=2016.963500,222.395500,-503.720300,90.647653,-0.183346,-0.000000
C02305=1927.753100,222.407300,-503.720300,90.647653,-0.183346,-0.000000
C02306=1936.624300,222.421800,-503.720300,90.647653,-0.183346,-0.000000
C02307=1941.897200,222.437700,-503.720300,90.647653,-0.183346,-0.000000
C02308=1915.919800,222.454300,-503.720300,90.647653,-0.183346,-0.000000
C02309=1941.539300,222.475200,-503.720300,90.647653,-0.183346,-0.000000
C02310=1969.735800,222.506600,-503.720300,90.647653,-0.183346,-0.000000
C02311=1958.400500,222.542400,-503.720300,90.647653,-0.183346,-0.000000
C02312=1952.915100,222.559000,-503.720300,90.647653,-0.183346,-0.000000
C02313=1927.316500,222.576200,-503.720300,90.647653,-0.183346,-0.000000
C02314=1935.896700,222.598500,-503.720300,90.647653,-0.183346,-0.000000
C02315=1927.083400,222.622300,-503.720300,90.647653,-0.183346,-0.000000
C02316=1971.501900,222.663700,-503.720300,90.647653,-0.183346,-0.000000
C02317=1985.419500,222.704600,-503.720300,90.647653,-0.183346,-0.000000
C02318=1933.249300,222.721700,-503.720300,90.647653,-0.183346,-0.000000
C02319=1983.244600,222.757300,-503.720300,90.647653,-0.183346,-0.000000
C02320=1966.958500,222.772500,-503.720300,90.647653,-0.183346,-0.000000
C02321=1971.033000,222.798900,-503.720300,90.647653,-0.183346,-0.000000
C02322=1977.908800,222.826200,-503.720300,90.647653,-0.183346,-0.000000
C02323=1956.249600,222.922500,-503.720300,90.647653,-0.183346,-0.000000
C02324=1963.733300,222.913400,-553.720300,90.647653,-0.183346,-0.000000
C02325=1956.256400,222.869900,-553.720300,90.647653,-0.183346,-0.000000
C02326=1948.604000,222.845500,-553.720300,90.647653,-0.183346,-0.000000
C02327=1964.013100,222.822500,-553.720300,90.647653,-0.183346,-0.000000
C02328=1979.543200,222.774200,-553.720300,90.647653,-0.183346,-0.000000
C02329=1979.134100,222.749900,-553.720300,90.647653,-0.183346,-0.000000
C02330=1991.483000,222.727900,-553.720300,90.647653,-0.183346,-0.000000
C02331=1961.051700,222.704900,-553.720300,90.647653,-0.183346,-0.000000
C02332=1983.390700,222.687000,-553.720300,90.647653,-0.183346,-0.000000
C02333=1962.251800,222.672200,-553.720300,90.647653,-0.183346,-0.000000
C02334=1991.225300,222.657800,-553.720300,90.647653,-0.183346,-0.000000
C02335=1934.904000,222.641100,-553.720300,90.647653,-0.183346,-0.000000
C02336=1988.588400,222.620800,-553.720300,90.647653,-0.183346,-0.000000
C02337=1998.476900,222.598500,-553.720300,90.647653,-0.183346,-0.000000
C02338=1957.514900,222.571500,-553.720300,90.647653,-0.183346,-0.000000
C02339=1957.921300,222.564100,-553.720300,90.647653,-0.183346,-0.000000
C02340=1912.022000,222.532600,-553.720300,90.647653,-0.183346,-0.000000
C02341=1993.708100,222.513500,-553.720300,90.647653,-0.183346,-0.000000
C02342=1980.501700,222.486700,-553.720300,90.647653,-0.183346,-0.000000
C02343=2004.291600,222.467100,-553.720300,90.647653,-0.183346,-0.000000
C02344=2002.901100,222.429600,-553.720300,90.647653,-0.183346,-0.000000
C02345=1951.911100,222.405600,-553.720300,90.647653,-0.183346,-0.000000
C02346=1909.620200,222.382000,-553.720300,90.647653,-0.183346,-0.000000
C02347=2014.840700,222.354300,-553.720300,90.647653,-0.183346,-0.000000
C02348=1937.761000,222.328200,-553.720300,90.647653,-0.183346,-0.000000
C02349=2012.811300,222.311000,-553.720300,90.647653,-0.183346,-0.000000
C02350=2018.822700,222.295100,-553.720300,90.647653,-0.183346,-0.000000
C02351=2008.094800,222.273400,-553.720300,90.647653,-0.183346,-0.000000
C02352=2018.441800,222.225200,-553.720300,90.647653,-0.183346,-0.000000
C02353=1978.897600,222.202900,-553.720300,90.647653,-0.183346,-0.000000
C02354=2016.124000,222.171500,-553.720300,90.647653,-0.183346,-0.000000
C02355=2005.897700,222.142900,-553.720300,90.647653,-0.183346,-0.000000
C02356=2029.998400,222.122200,-553.720300,90.647653,-0.183346,-0.000000
C02357=1889.817200,222.071100,-553.720300,90.647653,-0.183346,-0.000000
C02358=1897.116500,222.048200,-553.720300,90.647653,-0.183346,-0.000000
C02359=2045.315900,222.023500,-553.720300,90.647653,-0.183346,-0.000000
C02360=2045.517400,221.969400,-553.720300,90.647653,-0.183346,-0.000000
C02361=2037.969300,221.948700,-553.720300,90.647653,-0.183346,-0.000000
C02362=2042.005100,221.933300,-553.720300,90.647653,-0.183346,-0.000000
C02363=1898.029600,221.918400,-553.720300,90.647653,-0.183346,-0.000000
C02364=2032.408200,221.886400,-553.720300,90.647653,-0.183346,-0.000000
C02365=2014.803100,221.843400,-553.720300,90.647653,-0.183346,-0.000000
C02366=1897.770300,221.804200,-553.720300,90.647653,-0.183346,-0.000000
C02367=1893.088300,221.770800,-553.720300,90.647653,-0.183346,-0.000000
C02368=1880.302600,221.726500,-553.720300,90.647653,-0.183346,-0.000000
C02369=2046.366100,221.710000,-553.720300,90.647653,-0.183346,-0.000000
C02370=2069.403600,221.678900,-553.720300,90.647653,-0.183346,-0.000000
C02371=2040.087000,221.660000,-553.720300,90.647653,-0.183346,-0.000000
C02372=2051.630500,221.628600,-553.720300,90.647653,-0.183346,-0.000000
C02373=1875.490600,221.580900,-553.720300,90.647653,-0.183346,-0.000000
C02374=2081.618900,221.575900,-553.720300,90.647653,-0.183346,-0.000000
C02375=1798.549200,221.545800,-553.720300,90.647653,-0.183346,-0.000000
C02376=1860.471100,221.529600,-553.720300,90.647653,-0.183346,-0.000000
C02377=2089.008500,221.520800,-553.720300,90.647653,-0.183346,-0.000000
C02378=1867.309900,221.511000,-553.720300,90.647653,-0.183346,-0.000000
C02379=1802.747400,221.497100,-553.720300,90.647653,-0.183346,-0.000000
C02380=1795.578900,221.489200,-553.720300,90.647653,-0.183346,-0.000000
C02381=1850.696100,221.472100,-553.720300,90.647653,-0.183346,-0.000000
C02382=2071.297600,221.442400,-553.720300,90.647653,-0.183346,-0.000000
C02383=2066.326200,221.421100,-553.720300,90.647653,-0.183346,-0.000000
C02384=2185.271900,221.405200,-553.720300,90.647653,-0.183346,-0.000000
C02385=1808.383400,221.397800,-553.720300,90.647653,-0.183346,-0.000000
C02386=1860.874300,221.387300,-553.720300,90.647653,-0.183346,-0.000000
C02387=1793.872400,221.377500,-553.720300,90.647653,-0.183346,-0.000000
C02388=2058.125000,221.365200,-553.720300,90.647653,-0.183346,-0.000000
C02389=2171.695000,221.356300,-553.720300,90.647653,-0.183346,-0.000000
C02390=2051.746200,221.346500,-553.720300,90.647653,-0.183346,-0.000000
C02391=1831.047900,221.339700,-553.720300,90.647653,-0.183346,-0.000000
C02392=1805.769300,221.329900,-553.720300,90.647653,-0.183346,-0.000000
C02393=2093.721600,221.321800,-553.720300,90.647653,-0.183346,-0.000000
C02394=1829.779200,221.302500,-553.720300,90.647653,-0.183346,-0.000000
C02395=2095.057900,221.292100,-553.720300,90.647653,-0.183346,-0.000000
C02396=1835.604400,221.281600,-553.720300,90.647653,-0.183346,-0.000000
C02397=2176.560400,221.272500,-553.720300,90.647653,-0.183346,-0.000000
C02398=2070.281500,221.251200,-553.720300,90.647653,-0.183346,-0.000000
C02399=2177.772600,221.243400,-553.720300,90.647653,-0.183346,-0.000000
C02400=1859.955200,221.238000,-553.720300,90.647653,-0.183346,-0.000000
C02401=2154.924400,221.224500,-553.720300,90.647653,-0.183346,-0.000000
C02402=1849.898000,221.202500,-553.720300,90.647653,-0.183346,-0.000000
C02403=1794.349200,221.173500,-553.720300,90.647653,-0.183346,-0.000000
C02404=1827.378800,221.160300,-553.720300,90.647653,-0.183346,-0.000000
C02405=2164.964300,221.149200,-553.720300,90.647653,-0.183346,-0.000000
C02406=2170.479000,221.135300,-553.720300,90.647653,-0.183346,-0.000000
C02407=2089.777100,221.119400,-553.720300,90.647653,-0.183346,-0.000000
C02408=2079.439900,221.097800,-553.720300,90.647653,-0.183346,-0.000000
C02409=2162.975500,221.069800,-553.720300,90.647653,-0.183346,-0.000000
C02410=2079.119300,221.047800,-553.720300,90.647653,-0.183346,-0.000000
C02411=2103.256000,221.032900,-553.720300,90.647653,-0.183346,-0.000000
C02412=2172.854000,221.006900,-553.720300,90.647653,-0.183346,-0.000000
C02413=2096.169100,220.971500,-553.720300,90.647653,-0.183346,-0.000000
C02414=2115.178700,220.929600,-553.720300,90.647653,-0.183346,-0.000000
C02415=2172.080900,220.910600,-553.720300,90.647653,-0.183346,-0.000000
C02416=2165.845600,220.880100,-553.720300,90.647653,-0.183346,-0.000000
C02417=2102.209200,220.851200,-553.720300,90.647653,-0.183346,-0.000000
C02418=2158.791900,220.815400,-553.720300,90.647653,-0.183346,-0.000000
C02419=2124.265000,220.750200,-553.720300,90.647653,-0.183346,-0.000000
C02420=2146.776800,220.714700,-553.720300,90.647653,-0.183346,-0.000000
C02421=2123.652900,220.646800,-553.720300,90.647653,-0.183346,-0.000000
C02422=2154.536800,220.518100,-553.720300,90.647653,-0.183346,-0.000000
C02423=2135.182500,220.075100,-603.720300,90.647653,-0.183346,-0.000000
C02424=2155.869000,220.093700,-603.720300,90.647653,-0.183346,-0.000000
C02425=2141.886400,220.165200,-603.720300,90.647653,-0.183346,-0.000000
C02426=2153.492300,220.208900,-603.720300,90.647653,-0.183346,-0.000000
C02427=2118.162300,220.238300,-603.720300,90.647653,-0.183346,-0.000000
C02428=2076.220100,220.278500,-603.720300,90.647653,-0.183346,-0.000000
C02429=2112.488300,220.301200,-603.720300,90.647653,-0.183346,-0.000000
C02430=2143.693600,220.329900,-603.720300,90.647653,-0.183346,-0.000000
C02431=2060.873900,220.350500,-603.720300,90.647653,-0.183346,-0.000000
C02432=2072.706700,220.363300,-603.720300,90.647653,-0.183346,-0.000000
C02433=2166.622000,220.397400,-603.720300,90.647653,-0.183346,-0.000000
C02434=2134.801800,220.417400,-603.720300,90.647653,-0.183346,-0.000000
C02435=2108.284200,220.450500,-603.720300,90.647653,-0.183346,-0.000000
C02436=2166.981000,220.462000,-603.720300,90.647653,-0.183346,-0.000000
C02437=2072.248900,220.486300,-603.720300,90.647653,-0.183346,-0.000000
C02438=2170.151300,220.500800,-603.720300,90.647653,-0.183346,-0.000000
C02439=2120.281800,220.522500,-603.720300,90.647653,-0.183346,-0.000000
C02440=2089.470400,220.535300,-603.720300,90.647653,-0.183346,-0.000000
C02441=2054.688700,220.572100,-603.720300,90.647653,-0.183346,-0.000000
C02442=2155.004200,220.592000,-603.720300,90.647653,-0.183346,-0.000000
C02443=2081.393200,220.614300,-603.720300,90.647653,-0.183346,-0.000000
C02444=2165.525800,220.637300,-603.720300,90.647653,-0.183346,-0.000000
C02445=2093.464300,220.655600,-603.720300,90.647653,-0.183346,-0.000000
C02446=2069.170700,220.678500,-603.720300,90.647653,-0.183346,-0.000000
C02447=2178.378400,220.708300,-603.720300,90.647653,-0.183346,-0.000000
C02448=1873.645800,220.736300,-603.720300,90.647653,-0.183346,-0.000000
C02449=2167.297400,220.749100,-603.720300,90.647653,-0.183346,-0.000000
C02450=2070.704700,220.787300,-603.720300,90.647653,-0.183346,-0.000000
C02451=2025.783300,220.807600,-603.720300,90.647653,-0.183346,-0.000000
C02452=2038.907900,220.813000,-603.720300,90.647653,-0.183346,-0.000000
C02453=1845.141700,220.818400,-603.720300,90.647653,-0.183346,-0.000000
C02454=2098.071400,220.844100,-603.720300,90.647653,-0.183346,-0.000000
C02455=1834.488800,220.849800,-603.720300,90.647653,-0.183346,-0.000000
C02456=2182.059000,220.868400,-603.720300,90.647653,-0.183346,-0.000000
C02457=1826.858400,220.909300,-603.720300,90.647653,-0.183346,-0.000000
C02458=2008.883500,220.932900,-603.720300,90.647653,-0.183346,-0.000000
C02459=1827.799100,220.943400,-603.720300,90.647653,-0.183346,-0.000000
C02460=2189.484900,220.948500,-603.720300,90.647653,-0.183346,-0.000000
C02461=1825.755200,220.970100,-603.720300,90.647653,-0.183346,-0.000000
C02462=2172.874500,220.988300,-603.720300,90.647653,-0.183346,-0.000000
C02463=1861.689600,221.001200,-603.720300,90.647653,-0.183346,-0.000000
C02464=1902.491700,221.009300,-603.720300,90.647653,-0.183346,-0.000000
C02465=1896.399800,221.029200,-603.720300,90.647653,-0.183346,-0.000000
C02466=1842.596600,221.043700,-603.720300,90.647653,-0.183346,-0.000000
C02467=1821.337100,221.064700,-603.720300,90.647653,-0.183346,-0.000000
C02468=2040.053900,221.075800,-603.720300,90.647653,-0.183346,-0.000000
C02469=2030.334700,221.089700,-603.720300,90.647653,-0.183346,-0.000000
C02470=1921.654100,221.101500,-603.720300,90.647653,-0.183346,-0.000000
C02471=1913.056500,221.104600,-603.720300,90.647653,-0.183346,-0.000000
C02472=1815.721700,221.119800,-603.720300,90.647653,-0.183346,-0.000000
C02473=1892.427100,221.131900,-603.720300,90.647653,-0.183346,-0.000000
C02474=1855.127500,221.158600,-603.720300,90.647653,-0.183346,-0.000000
C02475=1812.770700,221.171100,-603.720300,90.647653,-0.183346,-0.000000
C02476=2041.204100,221.182300,-603.720300,90.647653,-0.183346,-0.000000
C02477=2185.732000,221.195800,-603.720300,90.647653,-0.183346,-0.000000
C02478=1929.095500,221.205600,-603.720300,90.647653,-0.183346,-0.000000
C02479=1833.140600,221.219800,-603.720300,90.647653,-0.183346,-0.000000
C02480=2020.116800,221.225500,-603.720300,90.647653,-0.183346,-0.000000
C02481=1883.750800,221.247500,-603.720300,90.647653,-0.183346,-0.000000
C02482=1897.924400,221.260000,-603.720300,90.647653,-0.183346,-0.000000
C02483=2014.324600,221.276900,-603.720300,90.647653,-0.183346,-0.000000
C02484=1908.464100,221.297800,-603.720300,90.647653,-0.183346,-0.000000
C02485=2003.540200,221.324800,-603.720300,90.647653,-0.183346,-0.000000
C02486=2006.842800,221.347500,-603.720300,90.647653,-0.183346,-0.000000
C02487=1886.125800,221.358300,-603.720300,90.647653,-0.183346,-0.000000
C02488=1870.093700,221.373100,-603.720300,90.647653,-0.183346,-0.000000
C02489=1933.986000,221.382600,-603.720300,90.647653,-0.183346,-0.000000
C02490=1959.483800,221.387300,-603.720300,90.647653,-0.183346,-0.000000
C02491=1798.584100,221.405600,-603.720300,90.647653,-0.183346,-0.000000
C02492=2016.296900,221.445100,-603.720300,90.647653,-0.183346,-0.000000
C02493=1972.695500,221.459600,-603.720300,90.647653,-0.183346,-0.000000
C02494=1986.916100,221.479900,-603.720300,90.647653,-0.183346,-0.000000
C02495=1944.214700,221.487700,-603.720300,90.647653,-0.183346,-0.000000
C02496=1886.406000,221.531600,-603.720300,90.647653,-0.183346,-0.000000
C02497=1896.365700,221.585300,-603.720300,90.647653,-0.183346,-0.000000
C02498=2035.527700,221.603600,-603.720300,90.647653,-0.183346,-0.000000
C02499=1926.518400,221.650200,-603.720300,90.647653,-0.183346,-0.000000
C02500=1903.812700,221.675500,-603.720300,90.647653,-0.183346,-0.000000
C02501=1922.073000,221.693400,-603.720300,90.647653,-0.183346,-0.000000
C02502=2009.734500,221.713400,-603.720300,90.647653,-0.183346,-0.000000
C02503=1993.013600,221.737000,-603.720300,90.647653,-0.183346,-0.000000
C02504=1987.631200,221.795100,-603.720300,90.647653,-0.183346,-0.000000
C02505=2019.393500,221.821800,-603.720300,90.647653,-0.183346,-0.000000
C02506=1973.778300,221.859300,-603.720300,90.647653,-0.183346,-0.000000
C02507=1934.952800,221.916700,-603.720300,90.647653,-0.183346,-0.000000
C02508=1994.054700,221.956300,-603.720300,90.647653,-0.183346,-0.000000
C02509=1977.630300,222.055300,-603.720300,90.647653,-0.183346,-0.000000
C02510=2001.389700,222.092900,-603.720300,90.647653,-0.183346,-0.000000
C02511=1961.318200,222.132300,-603.720300,90.647653,-0.183346,-0.000000
C02512=1967.736600,222.178100,-603.720300,90.647653,-0.183346,-0.000000
C02513=1994.900900,222.229600,-603.720300,90.647653,-0.183346,-0.000000
C02514=1959.228000,222.367100,-603.720300,90.647653,-0.183346,-0.000000
C02515=1799.111400,221.484600,-653.720300,90.647653,-0.183346,-0.000000
C02516=1797.016300,221.411200,-653.720300,90.647653,-0.183346,-0.000000
C02517=1797.597800,221.335600,-653.720300,90.647653,-0.183346,-0.000000
C02518=1812.527200,221.182900,-653.720300,90.647653,-0.183346,-0.000000
C02519=1808.531200,221.140000,-653.720300,90.647653,-0.183346,-0.000000
C02520=1794.828500,221.119800,-653.720300,90.647653,-0.183346,-0.000000
C02521=1818.252100,221.083300,-653.720300,90.647653,-0.183346,-0.000000
C02522=1939.426100,221.017100,-653.720300,90.647653,-0.183346,-0.000000
C02523=1794.174600,220.972800,-653.720300,90.647653,-0.183346,-0.000000
C02524=1920.488500,220.931900,-653.720300,90.647653,-0.183346,-0.000000
C02525=1993.501900,220.901200,-653.720300,90.647653,-0.183346,-0.000000
C02526=1906.745400,220.887000,-653.720300,90.647653,-0.183346,-0.000000
C02527=1821.826400,220.865400,-653.720300,90.647653,-0.183346,-0.000000
C02528=1952.228800,220.839700,-653.720300,90.647653,-0.183346,-0.000000
C02529=1899.610300,220.811300,-653.720300,90.647653,-0.183346,-0.000000
C02530=2005.113900,220.804600,-653.720300,90.647653,-0.183346,-0.000000
C02531=1920.095000,220.794400,-653.720300,90.647653,-0.183346,-0.000000
C02532=1993.508000,220.782600,-653.720300,90.647653,-0.183346,-0.000000
C02533=1964.485300,220.772000,-653.720300,90.647653,-0.183346,-0.000000
C02534=1960.437900,220.751500,-653.720300,90.647653,-0.183346,-0.000000
C02535=1944.239800,220.715000,-653.720300,90.647653,-0.183346,-0.000000
C02536=1860.805000,220.704200,-653.720300,90.647653,-0.183346,-0.000000
C02537=1876.569800,220.697300,-653.720300,90.647653,-0.183346,-0.000000
C02538=1851.373000,220.686300,-653.720300,90.647653,-0.183346,-0.000000
C02539=1848.454300,220.660600,-653.720300,90.647653,-0.183346,-0.000000
C02540=2185.567200,220.634300,-653.720300,90.647653,-0.183346,-0.000000
C02541=1837.295200,220.622800,-653.720300,90.647653,-0.183346,-0.000000
C02542=2178.745800,220.608700,-653.720300,90.647653,-0.183346,-0.000000
C02543=2181.412100,220.596800,-653.720300,90.647653,-0.183346,-0.000000
C02544=1884.394900,220.590000,-653.720300,90.647653,-0.183346,-0.000000
C02545=1928.752500,220.581900,-653.720300,90.647653,-0.183346,-0.000000
C02546=1935.459600,220.557300,-653.720300,90.647653,-0.183346,-0.000000
C02547=1974.551600,220.544400,-653.720300,90.647653,-0.183346,-0.000000
C02548=1983.119600,220.533900,-653.720300,90.647653,-0.183346,-0.000000
C02549=1956.770000,220.518400,-653.720300,90.647653,-0.183346,-0.000000
C02550=2180.850600,220.504200,-653.720300,90.647653,-0.183346,-0.000000
C02551=2029.057400,220.497800,-653.720300,90.647653,-0.183346,-0.000000
C02552=2008.258900,220.473700,-653.720300,90.647653,-0.183346,-0.000000
C02553=1930.929900,220.451800,-653.720300,90.647653,-0.183346,-0.000000
C02554=1879.009900,220.439300,-653.720300,90.647653,-0.183346,-0.000000
C02555=2186.746100,220.425300,-653.720300,90.647653,-0.183346,-0.000000
C02556=1907.260200,220.400200,-653.720300,90.647653,-0.183346,-0.000000
C02557=2041.942000,220.386600,-653.720300,90.647653,-0.183346,-0.000000
C02558=1896.038400,220.367400,-653.720300,90.647653,-0.183346,-0.000000
C02559=1863.364000,220.361300,-653.720300,90.647653,-0.183346,-0.000000
C02560=2027.041600,220.353400,-653.720300,90.647653,-0.183346,-0.000000
C02561=2189.914900,220.338000,-653.720300,90.647653,-0.183346,-0.000000
C02562=1856.782800,220.321800,-653.720300,90.647653,-0.183346,-0.000000
C02563=1870.979700,220.312000,-653.720300,90.647653,-0.183346,-0.000000
C02564=2172.182300,220.292800,-653.720300,90.647653,-0.183346,-0.000000
C02565=2168.310300,220.290000,-653.720300,90.647653,-0.183346,-0.000000
C02566=1916.132400,220.277200,-653.720300,90.647653,-0.183346,-0.000000
C02567=1898.895400,220.267000,-653.720300,90.647653,-0.183346,-0.000000
C02568=2021.451000,220.242700,-653.720300,90.647653,-0.183346,-0.000000
C02569=1961.960700,220.226200,-653.720300,90.647653,-0.183346,-0.000000
C02570=1931.745800,220.200100,-653.720300,90.647653,-0.183346,-0.000000
C02571=2016.990100,220.187600,-653.720300,90.647653,-0.183346,-0.000000
C02572=2167.245900,220.170400,-653.720300,90.647653,-0.183346,-0.000000
C02573=1877.351100,220.147400,-653.720300,90.647653,-0.183346,-0.000000
C02574=2037.722500,220.133400,-653.720300,90.647653,-0.183346,-0.000000
C02575=2079.880500,220.105900,-653.720300,90.647653,-0.183346,-0.000000
C02576=1931.420000,220.095100,-653.720300,90.647653,-0.183346,-0.000000
C02577=2071.825900,220.079200,-653.720300,90.647653,-0.183346,-0.000000
C02578=2164.985500,220.068000,-653.720300,90.647653,-0.183346,-0.000000
C02579=2065.291400,220.056600,-653.720300,90.647653,-0.183346,-0.000000
C02580=2147.782700,220.034900,-653.720300,90.647653,-0.183346,-0.000000
C02581=2048.202900,220.018000,-653.720300,90.647653,-0.183346,-0.000000
C02582=2151.836000,220.001500,-653.720300,90.647653,-0.183346,-0.000000
C02583=2149.211400,219.992000,-653.720300,90.647653,-0.183346,-0.000000
C02584=1969.603600,219.976200,-653.720300,90.647653,-0.183346,-0.000000
C02585=2062.163300,219.956700,-653.720300,90.647653,-0.183346,-0.000000
C02586=2095.969300,219.936600,-653.720300,90.647653,-0.183346,-0.000000
C02587=2073.497600,219.921100,-653.720300,90.647653,-0.183346,-0.000000
C02588=2129.535300,219.898500,-653.720300,90.647653,-0.183346,-0.000000
C02589=2161.709600,219.890700,-653.720300,90.647653,-0.183346,-0.000000
C02590=2086.631100,219.869400,-653.720300,90.647653,-0.183346,-0.000000
C02591=2156.454500,219.857900,-653.720300,90.647653,-0.183346,-0.000000
C02592=2072.521600,219.846800,-653.720300,90.647653,-0.183346,-0.000000
C02593=2141.120300,219.833600,-653.720300,90.647653,-0.183346,-0.000000
C02594=2160.733600,219.824100,-653.720300,90.647653,-0.183346,-0.000000
C02595=2027.707100,219.810900,-653.720300,90.647653,-0.183346,-0.000000
C02596=2092.652900,219.784300,-653.720300,90.647653,-0.183346,-0.000000
C02597=2123.747400,219.769100,-653.720300,90.647653,-0.183346,-0.000000
C02598=2153.192500,219.750500,-653.720300,90.647653,-0.183346,-0.000000
C02599=2092.906200,219.742500,-653.720300,90.647653,-0.183346,-0.000000
C02600=2123.769700,219.725100,-653.720300,90.647653,-0.183346,-0.000000
C02601=2083.229300,219.685600,-653.720300,90.647653,-0.183346,-0.000000
C02602=2126.587000,219.667400,-653.720300,90.647653,-0.183346,-0.000000
C02603=2134.480500,219.652500,-653.720300,90.647653,-0.183346,-0.000000
C02604=2101.138600,219.638300,-653.720300,90.647653,-0.183346,-0.000000
C02605=2117.690700,219.611600,-653.720300,90.647653,-0.183346,-0.000000
C02606=2115.842700,219.590700,-653.720300,90.647653,-0.183346,-0.000000
C02607=2127.919800,219.557600,-653.720300,90.647653,-0.183346,-0.000000
C02608=2113.565000,219.512000,-653.720300,90.647653,-0.183346,-0.000000
C02609=2072.715400,218.998100,-703.720300,90.647653,-0.183346,-0.000000
C02610=2063.281400,219.120700,-703.720300,90.647653,-0.183346,-0.000000
C02611=2093.116500,219.165700,-703.720300,90.647653,-0.183346,-0.000000
C02612=2076.539300,219.191300,-703.720300,90.647653,-0.183346,-0.000000
C02613=2088.785800,219.224800,-703.720300,90.647653,-0.183346,-0.000000
C02614=1995.233700,219.244700,-703.720300,90.647653,-0.183346,-0.000000
C02615=2081.333600,219.255200,-703.720300,90.647653,-0.183346,-0.000000
C02616=2022.588900,219.269700,-703.720300,90.647653,-0.183346,-0.000000
C02617=2028.734200,219.280200,-703.720300,90.647653,-0.183346,-0.000000
C02618=1977.350800,219.289300,-703.720300,90.647653,-0.183346,-0.000000
C02619=2106.833500,219.311300,-703.720300,90.647653,-0.183346,-0.000000
C02620=2116.884200,219.322100,-703.720300,90.647653,-0.183346,-0.000000
C02621=2012.897300,219.332900,-703.720300,90.647653,-0.183346,-0.000000
C02622=2059.388800,219.340300,-703.720300,90.647653,-0.183346,-0.000000
C02623=2047.652200,219.353500,-703.720300,90.647653,-0.183346,-0.000000
C02624=2082.861600,219.357600,-703.720300,90.647653,-0.183346,-0.000000
C02625=2037.173500,219.371400,-703.720300,90.647653,-0.183346,-0.000000
C02626=2099.311500,219.384200,-703.720300,90.647653,-0.183346,-0.000000
C02627=2039.965100,219.399100,-703.720300,90.647653,-0.183346,-0.000000
C02628=1981.559000,219.413600,-703.720300,90.647653,-0.183346,-0.000000
C02629=2065.638900,219.420100,-703.720300,90.647653,-0.183346,-0.000000
C02630=2130.302100,219.430200,-703.720300,90.647653,-0.183346,-0.000000
C02631=2124.640700,219.441300,-703.720300,90.647653,-0.183346,-0.000000
C02632=2075.078200,219.456200,-703.720300,90.647653,-0.183346,-0.000000
C02633=2042.197800,219.467000,-703.720300,90.647653,-0.183346,-0.000000
C02634=2068.814900,219.477200,-703.720300,90.647653,-0.183346,-0.000000
C02635=2058.284300,219.485900,-703.720300,90.647653,-0.183346,-0.000000
C02636=2057.105500,219.495400,-703.720300,90.647653,-0.183346,-0.000000
C02637=2133.991800,219.502500,-703.720300,90.647653,-0.183346,-0.000000
C02638=2007.174500,219.516300,-703.720300,90.647653,-0.183346,-0.000000
C02639=2120.815400,219.522800,-703.720300,90.647653,-0.183346,-0.000000
C02640=2139.440300,219.536600,-703.720300,90.647653,-0.183346,-0.000000
C02641=2047.526900,219.549800,-703.720300,90.647653,-0.183346,-0.000000
C02642=2190.491800,219.570400,-703.720300,90.647653,-0.183346,-0.000000
C02643=2133.701500,219.580200,-703.720300,90.647653,-0.183346,-0.000000
C02644=2149.100600,219.605200,-703.720300,90.647653,-0.183346,-0.000000
C02645=2145.670200,219.611300,-703.720300,90.647653,-0.183346,-0.000000
C02646=2153.555700,219.622400,-703.720300,90.647653,-0.183346,-0.000000
C02647=2156.072900,219.636300,-703.720300,90.647653,-0.183346,-0.000000
C02648=1911.271200,219.646400,-703.720300,90.647653,-0.183346,-0.000000
C02649=1996.980700,219.658900,-703.720300,90.647653,-0.183346,-0.000000
C02650=1962.517400,219.669200,-703.720300,90.647653,-0.183346,-0.000000
C02651=2019.679000,219.674500,-703.720300,90.647653,-0.183346,-0.000000
C02652=2151.272000,219.686600,-703.720300,90.647653,-0.183346,-0.000000
C02653=1978.235100,219.697800,-703.720300,90.647653,-0.183346,-0.000000
C02654=2190.653100,219.710900,-703.720300,90.647653,-0.183346,-0.000000
C02655=2162.636300,219.719700,-703.720300,90.647653,-0.183346,-0.000000
C02656=1903.307700,219.746800,-703.720300,90.647653,-0.183346,-0.000000
C02657=1940.427800,219.762600,-703.720300,90.647653,-0.183346,-0.000000
C02658=2183.514100,219.779600,-703.720300,90.647653,-0.183346,-0.000000
C02659=1959.607500,219.797400,-703.720300,90.647653,-0.183346,-0.000000
C02660=1883.120600,219.817700,-703.720300,90.647653,-0.183346,-0.000000
C02661=1912.425600,219.835900,-703.720300,90.647653,-0.183346,-0.000000
C02662=2178.141400,219.849700,-703.720300,90.647653,-0.183346,-0.000000
C02663=2024.153600,219.862300,-703.720300,90.647653,-0.183346,-0.000000
C02664=2178.001600,219.875100,-703.720300,90.647653,-0.183346,-0.000000
C02665=2183.166400,219.887600,-703.720300,90.647653,-0.183346,-0.000000
C02666=2174.232800,219.909900,-703.720300,90.647653,-0.183346,-0.000000
C02667=1897.447600,219.915700,-703.720300,90.647653,-0.183346,-0.000000
C02668=1932.657600,219.930900,-703.720300,90.647653,-0.183346,-0.000000
C02669=1878.214800,219.966000,-703.720300,90.647653,-0.183346,-0.000000
C02670=1895.386600,219.986000,-703.720300,90.647653,-0.183346,-0.000000
